LIN {X 0,Y 206.643,Z 558.739,A -85,B 0,C 180,E1 -21191.562,E2 -21191.562} C_VEL
LIN {X 0,Y 206.656,Z 558.72,A -85,B 0,C 180,E1 -21195.573,E2 -21195.573} C_VEL
LIN {X 0,Y 206.699,Z 558.712,A -85,B 0,C 180,E1 -21199.757,E2 -21199.757} C_VEL
LIN {X 0,Y 206.719,Z 558.701,A -85,B 0,C 180,E1 -21202.268,E2 -21202.268} C_VEL
LIN {X 0,Y 206.705,Z 558.728,A -85,B 0,C 180,E1 -21207.043,E2 -21207.043} C_VEL
LIN {X 0,Y 206.761,Z 558.716,A -85,B 0,C 180,E1 -21212.095,E2 -21212.095} C_VEL
LIN {X 0,Y 206.78,Z 558.717,A -85,B 0,C 180,E1 -21216.583,E2 -21216.583} C_VEL
LIN {X 0,Y 206.87,Z 558.707,A -85,B 0,C 180,E1 -21222.196,E2 -21222.196} C_VEL
LIN {X 0,Y 206.907,Z 558.71,A -85,B 0,C 180,E1 -21226.245,E2 -21226.245} C_VEL
LIN {X 0,Y 207.099,Z 558.667,A -85,B 0,C 180,E1 -21230.231,E2 -21230.231} C_VEL
LIN {X 0,Y 207.172,Z 558.672,A -85,B 0,C 180,E1 -21232.201,E2 -21232.201} C_VEL
LIN {X 0,Y 207.376,Z 558.637,A -85,B 0,C 180,E1 -21238.058,E2 -21238.058} C_VEL
LIN {X 0,Y 207.513,Z 558.637,A -85,B 0,C 180,E1 -21240,E2 -21240} C_VEL
LIN {X 0,Y 207.08,Z 558.67,A -85,B 0,C 180,E1 -21243.892,E2 -21243.892} C_VEL
LIN {X 0,Y 207.182,Z 558.674,A -85,B 0,C 180,E1 -21247.798,E2 -21247.798} C_VEL
LIN {X 0,Y 206.977,Z 558.693,A -85,B 0,C 180,E1 -21251.755,E2 -21251.755} C_VEL
LIN {X 0,Y 206.86,Z 558.701,A -85,B 0,C 180,E1 -21255.771,E2 -21255.771} C_VEL
LIN {X 0,Y 206.793,Z 558.723,A -85,B 0,C 180,E1 -21259.868,E2 -21259.868} C_VEL
LIN {X 0,Y 206.757,Z 558.732,A -85,B 0,C 180,E1 -21264.073,E2 -21264.073} C_VEL
LIN {X 0,Y 206.731,Z 558.734,A -85,B 0,C 180,E1 -21268.421,E2 -21268.421} C_VEL
LIN {X 0,Y 206.693,Z 558.739,A -85,B 0,C 180,E1 -21272.959,E2 -21272.959} C_VEL
LIN {X 0,Y 206.658,Z 558.711,A -85,B 0,C 180,E1 -21276.382,E2 -21276.382} C_VEL
LIN {X 0,Y 205.988,Z 558.801,A -85,B 0,C 180,E1 -21277.465,E2 -21277.465} C_VEL
LIN {X 0,Y 203.169,Z 559.171,A -85,B 0,C 180,E1 -21279.168,E2 -21279.168} C_VEL
LIN {X 0,Y 200.309,Z 559.522,A -85,B 0,C 180,E1 -21280.916,E2 -21280.916} C_VEL
LIN {X 0,Y 199.623,Z 559.597,A -85,B 0,C 180,E1 -21282.051,E2 -21282.051} C_VEL
LIN {X 0,Y 199.665,Z 559.81,A -85,B 0,C 180,E1 -21283.274,E2 -21283.274} C_VEL
LIN {X 0,Y 201.361,Z 565.662,A -85,B 0,C 180,E1 -21286.98,E2 -21286.98} C_VEL
LIN {X 0,Y 203.872,Z 570.231,A -85,B 0,C 180,E1 -21287.939,E2 -21287.939} C_VEL
LIN {X 0,Y 209.554,Z 580.486,A -85,B 0,C 180,E1 -21289.769,E2 -21289.769} C_VEL
LIN {X 0,Y 215.631,Z 592.995,A -85,B 0,C 180,E1 -21291.634,E2 -21291.634} C_VEL
LIN {X 0,Y 221.774,Z 607.312,A -85,B 0,C 180,E1 -21293.438,E2 -21293.438} C_VEL
LIN {X 0,Y 222.893,Z 610.666,A -85,B 0,C 180,E1 -21293.781,E2 -21293.781} C_VEL
LIN {X 0,Y 224.518,Z 623.901,A -85,B 0,C 180,E1 -21294.591,E2 -21294.591} C_VEL
LIN {X 0,Y 222.125,Z 674.384,A -85,B 0,C 180,E1 -21296.151,E2 -21296.151} C_VEL
LIN {X 0,Y 220.762,Z 687.705,A -85,B 0,C 180,E1 -21296.878,E2 -21296.878} C_VEL
LIN {X 0,Y 218.764,Z 699.996,A -85,B 0,C 180,E1 -21297.856,E2 -21297.856} C_VEL
LIN {X 0,Y 216.36,Z 712.201,A -85,B 0,C 180,E1 -21299.231,E2 -21299.231} C_VEL
LIN {X 0,Y 213.518,Z 723.76,A -85,B 0,C 180,E1 -21300.957,E2 -21300.957} C_VEL
LIN {X 0,Y 210.646,Z 734.172,A -85,B 0,C 180,E1 -21302.964,E2 -21302.964} C_VEL
LIN {X 0,Y 208.011,Z 742.689,A -85,B 0,C 180,E1 -21305.02,E2 -21305.02} C_VEL
LIN {X 0,Y 205.094,Z 751.926,A -85,B 0,C 180,E1 -21307.858,E2 -21307.858} C_VEL
LIN {X 0,Y 202.534,Z 759.353,A -85,B 0,C 180,E1 -21310.754,E2 -21310.754} C_VEL
LIN {X 0,Y 200.516,Z 765.318,A -85,B 0,C 180,E1 -21313.718,E2 -21313.718} C_VEL
LIN {X 0,Y 199.003,Z 770.036,A -85,B 0,C 180,E1 -21316.731,E2 -21316.731} C_VEL
LIN {X 0,Y 198.024,Z 773.649,A -85,B 0,C 180,E1 -21319.78,E2 -21319.78} C_VEL
LIN {X 0,Y 197.589,Z 775.512,A -85,B 0,C 180,E1 -21321.822,E2 -21321.822} C_VEL
LIN {X 0,Y 197.34,Z 776.909,A -85,B 0,C 180,E1 -21323.869,E2 -21323.869} C_VEL
LIN {X 0,Y 197.247,Z 778.517,A -85,B 0,C 180,E1 -21327.96,E2 -21327.96} C_VEL
LIN {X 0,Y 197.331,Z 778.731,A -85,B 0,C 180,E1 -21330.002,E2 -21330.002} C_VEL
LIN {X 0,Y 197.378,Z 778.507,A -85,B 0,C 180,E1 -21332.042,E2 -21332.042} C_VEL
LIN {X 0,Y 197.753,Z 777.534,A -85,B 0,C 180,E1 -21335.265,E2 -21335.265} C_VEL
LIN {X 0,Y 198.038,Z 780.359,A -85,B 0,C 180,E1 -21338.163,E2 -21338.163} C_VEL
LIN {X 0,Y 198.542,Z 781.793,A -85,B 0,C 180,E1 -21340.196,E2 -21340.196} C_VEL
LIN {X 0,Y 199.412,Z 782.694,A -85,B 0,C 180,E1 -21342.21,E2 -21342.21} C_VEL
LIN {X 0,Y 200.565,Z 783.037,A -85,B 0,C 180,E1 -21344.201,E2 -21344.201} C_VEL
LIN {X 0,Y 201.94,Z 782.915,A -85,B 0,C 180,E1 -21346.168,E2 -21346.168} C_VEL
LIN {X 0,Y 203.619,Z 782.336,A -85,B 0,C 180,E1 -21348.099,E2 -21348.099} C_VEL
LIN {X 0,Y 205.58,Z 781.284,A -85,B 0,C 180,E1 -21349.992,E2 -21349.992} C_VEL
LIN {X 0,Y 209.226,Z 778.633,A -85,B 0,C 180,E1 -21352.726,E2 -21352.726} C_VEL
LIN {X 0,Y 213.345,Z 774.775,A -85,B 0,C 180,E1 -21355.358,E2 -21355.358} C_VEL
LIN {X 0,Y 218.05,Z 769.669,A -85,B 0,C 180,E1 -21357.864,E2 -21357.864} C_VEL
LIN {X 0,Y 223.14,Z 762.876,A -85,B 0,C 180,E1 -21360.262,E2 -21360.262} C_VEL
LIN {X 0,Y 227.906,Z 755.838,A -85,B 0,C 180,E1 -21362.138,E2 -21362.138} C_VEL
LIN {X 0,Y 232.926,Z 747.036,A -85,B 0,C 180,E1 -21363.933,E2 -21363.933} C_VEL
LIN {X 0,Y 237.2,Z 738.413,A -85,B 0,C 180,E1 -21365.295,E2 -21365.295} C_VEL
LIN {X 0,Y 241.08,Z 729.19,A -85,B 0,C 180,E1 -21366.441,E2 -21366.441} C_VEL
LIN {X 0,Y 244.956,Z 717.42,A -85,B 0,C 180,E1 -21367.568,E2 -21367.568} C_VEL
LIN {X 0,Y 248.238,Z 704.464,A -85,B 0,C 180,E1 -21368.462,E2 -21368.462} C_VEL
LIN {X 0,Y 255.779,Z 670.421,A -85,B 0,C 180,E1 -21370.309,E2 -21370.309} C_VEL
LIN {X 0,Y 259.608,Z 653.752,A -85,B 0,C 180,E1 -21371.148,E2 -21371.148} C_VEL
LIN {X 0,Y 258.402,Z 653.739,A -85,B 0,C 180,E1 -21374.047,E2 -21374.047} C_VEL
LIN {X 0,Y 257.974,Z 655.742,A -85,B 0,C 180,E1 -21376.424,E2 -21376.424} C_VEL
LIN {X 0,Y 257.979,Z 658.123,A -85,B 0,C 180,E1 -21378.026,E2 -21378.026} C_VEL
LIN {X 0,Y 256.348,Z 670.35,A -85,B 0,C 180,E1 -21380.313,E2 -21380.313} C_VEL
LIN {X 0,Y 255.161,Z 681.627,A -85,B 0,C 180,E1 -21382.065,E2 -21382.065} C_VEL
LIN {X 0,Y 254.844,Z 684.003,A -85,B 0,C 180,E1 -21382.343,E2 -21382.343} C_VEL
LIN {X 0,Y 248.904,Z 711.445,A -85,B 0,C 180,E1 -21383.759,E2 -21383.759} C_VEL
LIN {X 0,Y 245.558,Z 722.701,A -85,B 0,C 180,E1 -21384.58,E2 -21384.58} C_VEL
LIN {X 0,Y 241.35,Z 733.582,A -85,B 0,C 180,E1 -21385.654,E2 -21385.654} C_VEL
LIN {X 0,Y 236.31,Z 744.211,A -85,B 0,C 180,E1 -21387.128,E2 -21387.128} C_VEL
LIN {X 0,Y 231.588,Z 752.59,A -85,B 0,C 180,E1 -21388.623,E2 -21388.623} C_VEL
LIN {X 0,Y 226.898,Z 759.605,A -85,B 0,C 180,E1 -21390.291,E2 -21390.291} C_VEL
LIN {X 0,Y 222.191,Z 765.752,A -85,B 0,C 180,E1 -21392.189,E2 -21392.189} C_VEL
LIN {X 0,Y 217.858,Z 770.669,A -85,B 0,C 180,E1 -21394.183,E2 -21394.183} C_VEL
LIN {X 0,Y 213.113,Z 775.192,A -85,B 0,C 180,E1 -21396.688,E2 -21396.688} C_VEL
LIN {X 0,Y 210.249,Z 777.424,A -85,B 0,C 180,E1 -21398.426,E2 -21398.426} C_VEL
LIN {X 0,Y 207.601,Z 779.05,A -85,B 0,C 180,E1 -21400.212,E2 -21400.212} C_VEL
LIN {X 0,Y 205.294,Z 780.132,A -85,B 0,C 180,E1 -21402.055,E2 -21402.055} C_VEL
LIN {X 0,Y 203.381,Z 780.726,A -85,B 0,C 180,E1 -21403.952,E2 -21403.952} C_VEL
LIN {X 0,Y 201.76,Z 780.834,A -85,B 0,C 180,E1 -21405.887,E2 -21405.887} C_VEL
LIN {X 0,Y 200.399,Z 780.44,A -85,B 0,C 180,E1 -21407.853,E2 -21407.853} C_VEL
LIN {X 0,Y 199.338,Z 779.484,A -85,B 0,C 180,E1 -21409.847,E2 -21409.847} C_VEL
LIN {X 0,Y 198.172,Z 776.715,A -85,B 0,C 180,E1 -21413.225,E2 -21413.225} C_VEL
LIN {X 0,Y 197.867,Z 773.43,A -85,B 0,C 180,E1 -21415.926,E2 -21415.926} C_VEL
LIN {X 0,Y 197.89,Z 768.393,A -85,B 0,C 180,E1 -21418.983,E2 -21418.983} C_VEL
LIN {X 0,Y 198.227,Z 761.55,A -85,B 0,C 180,E1 -21422.032,E2 -21422.032} C_VEL
LIN {X 0,Y 198.413,Z 755.716,A -85,B 0,C 180,E1 -21424.062,E2 -21424.062} C_VEL
LIN {X 0,Y 198.864,Z 747.227,A -85,B 0,C 180,E1 -21426.477,E2 -21426.477} C_VEL
LIN {X 0,Y 199.278,Z 738.663,A -85,B 0,C 180,E1 -21428.38,E2 -21428.38} C_VEL
LIN {X 0,Y 199.692,Z 728.558,A -85,B 0,C 180,E1 -21430.135,E2 -21430.135} C_VEL
LIN {X 0,Y 200.238,Z 717.043,A -85,B 0,C 180,E1 -21431.643,E2 -21431.643} C_VEL
LIN {X 0,Y 200.585,Z 705.7,A -85,B 0,C 180,E1 -21432.714,E2 -21432.714} C_VEL
LIN {X 0,Y 201.604,Z 660.067,A -85,B 0,C 180,E1 -21435.674,E2 -21435.674} C_VEL
LIN {X 0,Y 200.19,Z 633.11,A -85,B 0,C 180,E1 -21437.362,E2 -21437.362} C_VEL
LIN {X 0,Y 200.23,Z 631.57,A -85,B 0,C 180,E1 -21437.622,E2 -21437.622} C_VEL
LIN {X 0,Y 202.024,Z 611.253,A -85,B 0,C 180,E1 -21443.04,E2 -21443.04} C_VEL
LIN {X 0,Y 204.085,Z 591.489,A -85,B 0,C 180,E1 -21448.262,E2 -21448.262} C_VEL
LIN {X 0,Y 204.812,Z 584.337,A -85,B 0,C 180,E1 -21450.145,E2 -21450.145} C_VEL
LIN {X 0,Y 201.716,Z 569.092,A -85,B 0,C 180,E1 -21454.413,E2 -21454.413} C_VEL
LIN {X 0,Y 199.808,Z 559.78,A -85,B 0,C 180,E1 -21457.157,E2 -21457.157} C_VEL
LIN {X 0,Y 199.581,Z 559.561,A -85,B 0,C 180,E1 -21462.31,E2 -21462.31} C_VEL
LIN {X 0,Y 199.677,Z 559.818,A -85,B 0,C 180,E1 -21466.585,E2 -21466.585} C_VEL
LIN {X 0,Y 199.952,Z 560.952,A -85,B 0,C 180,E1 -21466.993,E2 -21466.993} C_VEL
LIN {X 0,Y 201.638,Z 563.728,A -85,B 0,C 180,E1 -21467.594,E2 -21467.594} C_VEL
LIN {X 0,Y 202.715,Z 565.008,A -85,B 0,C 180,E1 -21467.934,E2 -21467.934} C_VEL
LIN {X 0,Y 205.044,Z 568.455,A -85,B 0,C 180,E1 -21468.681,E2 -21468.681} C_VEL
LIN {X 0,Y 213.235,Z 581.719,A -85,B 0,C 180,E1 -21471.169,E2 -21471.169} C_VEL
LIN {X 0,Y 220.429,Z 596.663,A -85,B 0,C 180,E1 -21473.27,E2 -21473.27} C_VEL
LIN {X 0,Y 225.025,Z 607.882,A -85,B 0,C 180,E1 -21474.578,E2 -21474.578} C_VEL
LIN {X 0,Y 222.424,Z 664.276,A -85,B 0,C 180,E1 -21476.339,E2 -21476.339} C_VEL
LIN {X 0,Y 221.083,Z 677.457,A -85,B 0,C 180,E1 -21477.073,E2 -21477.073} C_VEL
LIN {X 0,Y 219.394,Z 689.53,A -85,B 0,C 180,E1 -21478.09,E2 -21478.09} C_VEL
LIN {X 0,Y 217.347,Z 700.817,A -85,B 0,C 180,E1 -21479.382,E2 -21479.382} C_VEL
LIN {X 0,Y 214.559,Z 712.45,A -85,B 0,C 180,E1 -21481.107,E2 -21481.107} C_VEL
LIN {X 0,Y 211.759,Z 722.896,A -85,B 0,C 180,E1 -21483.114,E2 -21483.114} C_VEL
LIN {X 0,Y 209.106,Z 732.051,A -85,B 0,C 180,E1 -21485.345,E2 -21485.345} C_VEL
LIN {X 0,Y 206.368,Z 740.665,A -85,B 0,C 180,E1 -21487.998,E2 -21487.998} C_VEL
LIN {X 0,Y 203.743,Z 748.068,A -85,B 0,C 180,E1 -21490.869,E2 -21490.869} C_VEL
LIN {X 0,Y 201.639,Z 754.008,A -85,B 0,C 180,E1 -21493.808,E2 -21493.808} C_VEL
LIN {X 0,Y 199.942,Z 758.7,A -85,B 0,C 180,E1 -21496.791,E2 -21496.791} C_VEL
LIN {X 0,Y 198.741,Z 762.283,A -85,B 0,C 180,E1 -21499.814,E2 -21499.814} C_VEL
LIN {X 0,Y 198.164,Z 764.133,A -85,B 0,C 180,E1 -21501.843,E2 -21501.843} C_VEL
LIN {X 0,Y 197.671,Z 765.903,A -85,B 0,C 180,E1 -21504.575,E2 -21504.575} C_VEL
LIN {X 0,Y 197.407,Z 767.121,A -85,B 0,C 180,E1 -21507.958,E2 -21507.958} C_VEL
LIN {X 0,Y 197.401,Z 767.348,A -85,B 0,C 180,E1 -21509.998,E2 -21509.998} C_VEL
LIN {X 0,Y 197.406,Z 767.155,A -85,B 0,C 180,E1 -21512.038,E2 -21512.038} C_VEL
LIN {X 0,Y 197.669,Z 765.987,A -85,B 0,C 180,E1 -21515.419,E2 -21515.419} C_VEL
LIN {X 0,Y 198.162,Z 764.251,A -85,B 0,C 180,E1 -21518.154,E2 -21518.154} C_VEL
LIN {X 0,Y 199.056,Z 761.381,A -85,B 0,C 180,E1 -21521.195,E2 -21521.195} C_VEL
LIN {X 0,Y 200.419,Z 757.487,A -85,B 0,C 180,E1 -21524.207,E2 -21524.207} C_VEL
LIN {X 0,Y 202.212,Z 752.468,A -85,B 0,C 180,E1 -21527.181,E2 -21527.181} C_VEL
LIN {X 0,Y 204.465,Z 746.143,A -85,B 0,C 180,E1 -21530.102,E2 -21530.102} C_VEL
LIN {X 0,Y 207.302,Z 738.221,A -85,B 0,C 180,E1 -21532.945,E2 -21532.945} C_VEL
LIN {X 0,Y 209.92,Z 729.627,A -85,B 0,C 180,E1 -21535.424,E2 -21535.424} C_VEL
LIN {X 0,Y 212.584,Z 720.302,A -85,B 0,C 180,E1 -21537.568,E2 -21537.568} C_VEL
LIN {X 0,Y 215.469,Z 709.206,A -85,B 0,C 180,E1 -21539.558,E2 -21539.558} C_VEL
LIN {X 0,Y 217.881,Z 698.322,A -85,B 0,C 180,E1 -21541.069,E2 -21541.069} C_VEL
LIN {X 0,Y 220.02,Z 686.282,A -85,B 0,C 180,E1 -21542.344,E2 -21542.344} C_VEL
LIN {X 0,Y 221.684,Z 673.728,A -85,B 0,C 180,E1 -21543.299,E2 -21543.299} C_VEL
LIN {X 0,Y 222.779,Z 660.908,A -85,B 0,C 180,E1 -21543.918,E2 -21543.918} C_VEL
LIN {X 0,Y 225.154,Z 608.113,A -85,B 0,C 180,E1 -21545.54,E2 -21545.54} C_VEL
LIN {X 0,Y 219.131,Z 593.766,A -85,B 0,C 180,E1 -21547.258,E2 -21547.258} C_VEL
LIN {X 0,Y 212.658,Z 580.606,A -85,B 0,C 180,E1 -21549.166,E2 -21549.166} C_VEL
LIN {X 0,Y 205.028,Z 568.468,A -85,B 0,C 180,E1 -21551.492,E2 -21551.492} C_VEL
LIN {X 0,Y 202.812,Z 565.309,A -85,B 0,C 180,E1 -21552.2,E2 -21552.2} C_VEL
LIN {X 0,Y 202.07,Z 564.19,A -85,B 0,C 180,E1 -21552.445,E2 -21552.445} C_VEL
LIN {X 0,Y 200.158,Z 561.683,A -85,B 0,C 180,E1 -21553.072,E2 -21553.072} C_VEL
LIN {X 0,Y 199.577,Z 559.608,A -85,B 0,C 180,E1 -21553.387,E2 -21553.387} C_VEL
LIN {X 0,Y 199.615,Z 559.621,A -85,B 0,C 180,E1 -21558.014,E2 -21558.014} C_VEL
LIN {X 0,Y 199.673,Z 559.577,A -85,B 0,C 180,E1 -21560.742,E2 -21560.742} C_VEL
LIN {X 0,Y 199.631,Z 559.619,A -85,B 0,C 180,E1 -21565.717,E2 -21565.717} C_VEL
LIN {X 0,Y 199.699,Z 559.6,A -85,B 0,C 180,E1 -21568.136,E2 -21568.136} C_VEL
LIN {X 0,Y 199.681,Z 559.598,A -85,B 0,C 180,E1 -21572.771,E2 -21572.771} C_VEL
LIN {X 0,Y 199.732,Z 559.59,A -85,B 0,C 180,E1 -21577.228,E2 -21577.228} C_VEL
LIN {X 0,Y 199.832,Z 559.587,A -85,B 0,C 180,E1 -21581.721,E2 -21581.721} C_VEL
LIN {X 0,Y 199.841,Z 559.584,A -85,B 0,C 180,E1 -21585.749,E2 -21585.749} C_VEL
LIN {X 0,Y 200.064,Z 559.543,A -85,B 0,C 180,E1 -21589.884,E2 -21589.884} C_VEL
LIN {X 0,Y 200.033,Z 559.567,A -85,B 0,C 180,E1 -21593.95,E2 -21593.95} C_VEL
LIN {X 0,Y 200.316,Z 559.516,A -85,B 0,C 180,E1 -21597.989,E2 -21597.989} C_VEL
LIN {X 0,Y 200.477,Z 559.514,A -85,B 0,C 180,E1 -21600,E2 -21600} C_VEL
LIN {X 0,Y 200.026,Z 559.549,A -85,B 0,C 180,E1 -21604.029,E2 -21604.029} C_VEL
LIN {X 0,Y 200.126,Z 559.552,A -85,B 0,C 180,E1 -21608.075,E2 -21608.075} C_VEL
LIN {X 0,Y 199.908,Z 559.577,A -85,B 0,C 180,E1 -21612.177,E2 -21612.177} C_VEL
LIN {X 0,Y 199.799,Z 559.58,A -85,B 0,C 180,E1 -21616.344,E2 -21616.344} C_VEL
LIN {X 0,Y 199.818,Z 559.594,A -85,B 0,C 180,E1 -21618.454,E2 -21618.454} C_VEL
LIN {X 0,Y 199.731,Z 559.605,A -85,B 0,C 180,E1 -21623.818,E2 -21623.818} C_VEL
LIN {X 0,Y 199.702,Z 559.608,A -85,B 0,C 180,E1 -21628.385,E2 -21628.385} C_VEL
LIN {X 0,Y 199.666,Z 559.611,A -85,B 0,C 180,E1 -21632.356,E2 -21632.356} C_VEL
LIN {X 0,Y 199.638,Z 559.584,A -85,B 0,C 180,E1 -21636.76,E2 -21636.76} C_VEL
LIN {X 0,Y 199.669,Z 559.61,A -85,B 0,C 180,E1 -21639.314,E2 -21639.314} C_VEL
LIN {X 0,Y 199.623,Z 559.597,A -85,B 0,C 180,E1 -21642.051,E2 -21642.051} C_VEL
LIN {X 0,Y 199.313,Z 560.282,A -85,B 0,C 180,E1 -21642.984,E2 -21642.984} C_VEL
LIN {X 0,Y 198.369,Z 562.793,A -85,B 0,C 180,E1 -21644.129,E2 -21644.129} C_VEL
LIN {X 0,Y 197.419,Z 566.85,A -85,B 0,C 180,E1 -21645.236,E2 -21645.236} C_VEL
LIN {X 0,Y 197.48,Z 570.795,A -85,B 0,C 180,E1 -21646.115,E2 -21646.115} C_VEL
LIN {X 0,Y 198.563,Z 573.421,A -85,B 0,C 180,E1 -21646.705,E2 -21646.705} C_VEL
LIN {X 0,Y 203.685,Z 582.425,A -85,B 0,C 180,E1 -21648.456,E2 -21648.456} C_VEL
LIN {X 0,Y 210.102,Z 595.374,A -85,B 0,C 180,E1 -21650.541,E2 -21650.541} C_VEL
LIN {X 0,Y 216.727,Z 611.183,A -85,B 0,C 180,E1 -21652.607,E2 -21652.607} C_VEL
LIN {X 0,Y 217.406,Z 613.834,A -85,B 0,C 180,E1 -21652.85,E2 -21652.85} C_VEL
LIN {X 0,Y 218.724,Z 624.414,A -85,B 0,C 180,E1 -21653.533,E2 -21653.533} C_VEL
LIN {X 0,Y 216.213,Z 675.123,A -85,B 0,C 180,E1 -21655.151,E2 -21655.151} C_VEL
LIN {X 0,Y 214.664,Z 688.967,A -85,B 0,C 180,E1 -21655.945,E2 -21655.945} C_VEL
LIN {X 0,Y 212.576,Z 700.905,A -85,B 0,C 180,E1 -21656.943,E2 -21656.943} C_VEL
LIN {X 0,Y 209.92,Z 713.586,A -85,B 0,C 180,E1 -21658.461,E2 -21658.461} C_VEL
LIN {X 0,Y 206.973,Z 724.852,A -85,B 0,C 180,E1 -21660.226,E2 -21660.226} C_VEL
LIN {X 0,Y 203.997,Z 735.005,A -85,B 0,C 180,E1 -21662.286,E2 -21662.286} C_VEL
LIN {X 0,Y 201.01,Z 744.156,A -85,B 0,C 180,E1 -21664.642,E2 -21664.642} C_VEL
LIN {X 0,Y 198.218,Z 752.585,A -85,B 0,C 180,E1 -21667.396,E2 -21667.396} C_VEL
LIN {X 0,Y 195.461,Z 760.265,A -85,B 0,C 180,E1 -21670.576,E2 -21670.576} C_VEL
LIN {X 0,Y 193.045,Z 766.806,A -85,B 0,C 180,E1 -21674.157,E2 -21674.157} C_VEL
LIN {X 0,Y 191.66,Z 771.143,A -85,B 0,C 180,E1 -21677.292,E2 -21677.292} C_VEL
LIN {X 0,Y 191.013,Z 773.445,A -85,B 0,C 180,E1 -21679.401,E2 -21679.401} C_VEL
LIN {X 0,Y 190.538,Z 775.307,A -85,B 0,C 180,E1 -21681.518,E2 -21681.518} C_VEL
LIN {X 0,Y 190.278,Z 776.705,A -85,B 0,C 180,E1 -21683.64,E2 -21683.64} C_VEL
LIN {X 0,Y 190.155,Z 778.312,A -85,B 0,C 180,E1 -21687.884,E2 -21687.884} C_VEL
LIN {X 0,Y 190.236,Z 778.526,A -85,B 0,C 180,E1 -21690.002,E2 -21690.002} C_VEL
LIN {X 0,Y 190.291,Z 778.302,A -85,B 0,C 180,E1 -21692.118,E2 -21692.118} C_VEL
LIN {X 0,Y 190.844,Z 777.039,A -85,B 0,C 180,E1 -21696.12,E2 -21696.12} C_VEL
LIN {X 0,Y 191.058,Z 779.447,A -85,B 0,C 180,E1 -21698.463,E2 -21698.463} C_VEL
LIN {X 0,Y 191.594,Z 781.043,A -85,B 0,C 180,E1 -21700.57,E2 -21700.57} C_VEL
LIN {X 0,Y 192.511,Z 782.153,A -85,B 0,C 180,E1 -21702.655,E2 -21702.655} C_VEL
LIN {X 0,Y 193.704,Z 782.81,A -85,B 0,C 180,E1 -21704.715,E2 -21704.715} C_VEL
LIN {X 0,Y 195.147,Z 783.008,A -85,B 0,C 180,E1 -21706.747,E2 -21706.747} C_VEL
LIN {X 0,Y 196.885,Z 782.666,A -85,B 0,C 180,E1 -21708.741,E2 -21708.741} C_VEL
LIN {X 0,Y 198.942,Z 781.819,A -85,B 0,C 180,E1 -21710.689,E2 -21710.689} C_VEL
LIN {X 0,Y 201.489,Z 780.484,A -85,B 0,C 180,E1 -21712.564,E2 -21712.564} C_VEL
LIN {X 0,Y 205.568,Z 777.591,A -85,B 0,C 180,E1 -21715.301,E2 -21715.301} C_VEL
LIN {X 0,Y 210.343,Z 773.457,A -85,B 0,C 180,E1 -21717.891,E2 -21717.891} C_VEL
LIN {X 0,Y 215.547,Z 767.896,A -85,B 0,C 180,E1 -21720.359,E2 -21720.359} C_VEL
LIN {X 0,Y 220.307,Z 762.035,A -85,B 0,C 180,E1 -21722.301,E2 -21722.301} C_VEL
LIN {X 0,Y 226.49,Z 753.294,A -85,B 0,C 180,E1 -21724.494,E2 -21724.494} C_VEL
LIN {X 0,Y 231.437,Z 744.927,A -85,B 0,C 180,E1 -21726.042,E2 -21726.042} C_VEL
LIN {X 0,Y 236.629,Z 734.698,A -85,B 0,C 180,E1 -21727.509,E2 -21727.509} C_VEL
LIN {X 0,Y 240.761,Z 724.592,A -85,B 0,C 180,E1 -21728.607,E2 -21728.607} C_VEL
LIN {X 0,Y 244.395,Z 713.469,A -85,B 0,C 180,E1 -21729.514,E2 -21729.514} C_VEL
LIN {X 0,Y 248.288,Z 697.651,A -85,B 0,C 180,E1 -21730.488,E2 -21730.488} C_VEL
LIN {X 0,Y 254.976,Z 669.376,A -85,B 0,C 180,E1 -21731.936,E2 -21731.936} C_VEL
LIN {X 0,Y 257.137,Z 660.432,A -85,B 0,C 180,E1 -21732.442,E2 -21732.442} C_VEL
LIN {X 0,Y 256.503,Z 660.855,A -85,B 0,C 180,E1 -21734.367,E2 -21734.367} C_VEL
LIN {X 0,Y 256.112,Z 663.035,A -85,B 0,C 180,E1 -21736.573,E2 -21736.573} C_VEL
LIN {X 0,Y 256.07,Z 663.953,A -85,B 0,C 180,E1 -21737.123,E2 -21737.123} C_VEL
LIN {X 0,Y 254.151,Z 675.571,A -85,B 0,C 180,E1 -21739.301,E2 -21739.301} C_VEL
LIN {X 0,Y 252.699,Z 685.678,A -85,B 0,C 180,E1 -21740.859,E2 -21740.859} C_VEL
LIN {X 0,Y 246.939,Z 711.044,A -85,B 0,C 180,E1 -21742.144,E2 -21742.144} C_VEL
LIN {X 0,Y 243.455,Z 722.275,A -85,B 0,C 180,E1 -21742.943,E2 -21742.943} C_VEL
LIN {X 0,Y 239.627,Z 731.754,A -85,B 0,C 180,E1 -21743.826,E2 -21743.826} C_VEL
LIN {X 0,Y 234.811,Z 741.897,A -85,B 0,C 180,E1 -21745.081,E2 -21745.081} C_VEL
LIN {X 0,Y 229.638,Z 750.729,A -85,B 0,C 180,E1 -21746.572,E2 -21746.572} C_VEL
LIN {X 0,Y 224.314,Z 758.556,A -85,B 0,C 180,E1 -21748.279,E2 -21748.279} C_VEL
LIN {X 0,Y 219.033,Z 765.044,A -85,B 0,C 180,E1 -21750.176,E2 -21750.176} C_VEL
LIN {X 0,Y 215.229,Z 769.152,A -85,B 0,C 180,E1 -21751.739,E2 -21751.739} C_VEL
LIN {X 0,Y 209.958,Z 774.044,A -85,B 0,C 180,E1 -21754.205,E2 -21754.205} C_VEL
LIN {X 0,Y 206.715,Z 776.508,A -85,B 0,C 180,E1 -21755.922,E2 -21755.922} C_VEL
LIN {X 0,Y 203.717,Z 778.405,A -85,B 0,C 180,E1 -21757.698,E2 -21757.698} C_VEL
LIN {X 0,Y 200.973,Z 779.797,A -85,B 0,C 180,E1 -21759.531,E2 -21759.531} C_VEL
LIN {X 0,Y 198.596,Z 780.66,A -85,B 0,C 180,E1 -21761.428,E2 -21761.428} C_VEL
LIN {X 0,Y 196.589,Z 780.953,A -85,B 0,C 180,E1 -21763.382,E2 -21763.382} C_VEL
LIN {X 0,Y 194.888,Z 780.736,A -85,B 0,C 180,E1 -21765.379,E2 -21765.379} C_VEL
LIN {X 0,Y 193.494,Z 780.049,A -85,B 0,C 180,E1 -21767.413,E2 -21767.413} C_VEL
LIN {X 0,Y 192.389,Z 778.886,A -85,B 0,C 180,E1 -21769.476,E2 -21769.476} C_VEL
LIN {X 0,Y 191.6,Z 777.235,A -85,B 0,C 180,E1 -21771.563,E2 -21771.563} C_VEL
LIN {X 0,Y 190.968,Z 773.747,A -85,B 0,C 180,E1 -21774.607,E2 -21774.607} C_VEL
LIN {X 0,Y 190.904,Z 768.638,A -85,B 0,C 180,E1 -21777.89,E2 -21777.89} C_VEL
LIN {X 0,Y 191.188,Z 762.049,A -85,B 0,C 180,E1 -21781.053,E2 -21781.053} C_VEL
LIN {X 0,Y 191.466,Z 756.372,A -85,B 0,C 180,E1 -21783.156,E2 -21783.156} C_VEL
LIN {X 0,Y 191.885,Z 747.559,A -85,B 0,C 180,E1 -21785.781,E2 -21785.781} C_VEL
LIN {X 0,Y 192.283,Z 738.777,A -85,B 0,C 180,E1 -21787.82,E2 -21787.82} C_VEL
LIN {X 0,Y 192.664,Z 729.114,A -85,B 0,C 180,E1 -21789.595,E2 -21789.595} C_VEL
LIN {X 0,Y 193.165,Z 718.19,A -85,B 0,C 180,E1 -21791.144,E2 -21791.144} C_VEL
LIN {X 0,Y 193.579,Z 706.742,A -85,B 0,C 180,E1 -21792.315,E2 -21792.315} C_VEL
LIN {X 0,Y 194.525,Z 659.858,A -85,B 0,C 180,E1 -21795.52,E2 -21795.52} C_VEL
LIN {X 0,Y 193.109,Z 633.055,A -85,B 0,C 180,E1 -21797.268,E2 -21797.268} C_VEL
LIN {X 0,Y 193.106,Z 631.825,A -85,B 0,C 180,E1 -21797.473,E2 -21797.473} C_VEL
LIN {X 0,Y 195.009,Z 610.41,A -85,B 0,C 180,E1 -21803.356,E2 -21803.356} C_VEL
LIN {X 0,Y 197.294,Z 589.517,A -85,B 0,C 180,E1 -21809.036,E2 -21809.036} C_VEL
LIN {X 0,Y 197.717,Z 584.862,A -85,B 0,C 180,E1 -21810.297,E2 -21810.297} C_VEL
LIN {X 0,Y 194.737,Z 570.374,A -85,B 0,C 180,E1 -21814.456,E2 -21814.456} C_VEL
LIN {X 0,Y 192.739,Z 560.681,A -85,B 0,C 180,E1 -21817.382,E2 -21817.382} C_VEL
LIN {X 0,Y 192.522,Z 560.439,A -85,B 0,C 180,E1 -21823.103,E2 -21823.103} C_VEL
LIN {X 0,Y 192.607,Z 560.793,A -85,B 0,C 180,E1 -21824.646,E2 -21824.646} C_VEL
LIN {X 0,Y 192.938,Z 561.931,A -85,B 0,C 180,E1 -21825.055,E2 -21825.055} C_VEL
LIN {X 0,Y 194.545,Z 564.576,A -85,B 0,C 180,E1 -21825.683,E2 -21825.683} C_VEL
LIN {X 0,Y 195.73,Z 565.827,A -85,B 0,C 180,E1 -21826.086,E2 -21826.086} C_VEL
LIN {X 0,Y 198.122,Z 569.451,A -85,B 0,C 180,E1 -21826.931,E2 -21826.931} C_VEL
LIN {X 0,Y 204.033,Z 578.563,A -85,B 0,C 180,E1 -21828.895,E2 -21828.895} C_VEL
LIN {X 0,Y 208.753,Z 586.374,A -85,B 0,C 180,E1 -21830.369,E2 -21830.369} C_VEL
LIN {X 0,Y 215.819,Z 601.464,A -85,B 0,C 180,E1 -21832.542,E2 -21832.542} C_VEL
LIN {X 0,Y 219.224,Z 609.857,A -85,B 0,C 180,E1 -21833.562,E2 -21833.562} C_VEL
LIN {X 0,Y 216.633,Z 663.621,A -85,B 0,C 180,E1 -21835.259,E2 -21835.259} C_VEL
LIN {X 0,Y 215.217,Z 677.201,A -85,B 0,C 180,E1 -21836.013,E2 -21836.013} C_VEL
LIN {X 0,Y 213.422,Z 689.741,A -85,B 0,C 180,E1 -21837.087,E2 -21837.087} C_VEL
LIN {X 0,Y 211.287,Z 701.026,A -85,B 0,C 180,E1 -21838.405,E2 -21838.405} C_VEL
LIN {X 0,Y 208.37,Z 712.659,A -85,B 0,C 180,E1 -21840.164,E2 -21840.164} C_VEL
LIN {X 0,Y 205.461,Z 723.104,A -85,B 0,C 180,E1 -21842.22,E2 -21842.22} C_VEL
LIN {X 0,Y 202.491,Z 732.809,A -85,B 0,C 180,E1 -21844.664,E2 -21844.664} C_VEL
LIN {X 0,Y 199.794,Z 740.872,A -85,B 0,C 180,E1 -21847.234,E2 -21847.234} C_VEL
LIN {X 0,Y 197.025,Z 748.276,A -85,B 0,C 180,E1 -21850.19,E2 -21850.19} C_VEL
LIN {X 0,Y 194.823,Z 754.215,A -85,B 0,C 180,E1 -21853.225,E2 -21853.225} C_VEL
LIN {X 0,Y 193.033,Z 758.906,A -85,B 0,C 180,E1 -21856.309,E2 -21856.309} C_VEL
LIN {X 0,Y 191.748,Z 762.489,A -85,B 0,C 180,E1 -21859.438,E2 -21859.438} C_VEL
LIN {X 0,Y 191.127,Z 764.339,A -85,B 0,C 180,E1 -21861.54,E2 -21861.54} C_VEL
LIN {X 0,Y 190.569,Z 766.285,A -85,B 0,C 180,E1 -21864.709,E2 -21864.709} C_VEL
LIN {X 0,Y 190.317,Z 767.325,A -85,B 0,C 180,E1 -21867.882,E2 -21867.882} C_VEL
LIN {X 0,Y 190.306,Z 767.553,A -85,B 0,C 180,E1 -21869.998,E2 -21869.998} C_VEL
LIN {X 0,Y 190.316,Z 767.36,A -85,B 0,C 180,E1 -21872.114,E2 -21872.114} C_VEL
LIN {X 0,Y 190.721,Z 765.81,A -85,B 0,C 180,E1 -21876.345,E2 -21876.345} C_VEL
LIN {X 0,Y 191.125,Z 764.455,A -85,B 0,C 180,E1 -21878.456,E2 -21878.456} C_VEL
LIN {X 0,Y 192.098,Z 761.585,A -85,B 0,C 180,E1 -21881.606,E2 -21881.606} C_VEL
LIN {X 0,Y 193.538,Z 757.691,A -85,B 0,C 180,E1 -21884.724,E2 -21884.724} C_VEL
LIN {X 0,Y 195.431,Z 752.671,A -85,B 0,C 180,E1 -21887.797,E2 -21887.797} C_VEL
LIN {X 0,Y 197.816,Z 746.346,A -85,B 0,C 180,E1 -21890.808,E2 -21890.808} C_VEL
LIN {X 0,Y 200.779,Z 738.424,A -85,B 0,C 180,E1 -21893.735,E2 -21893.735} C_VEL
LIN {X 0,Y 203.426,Z 730.126,A -85,B 0,C 180,E1 -21896.204,E2 -21896.204} C_VEL
LIN {X 0,Y 206.328,Z 720.502,A -85,B 0,C 180,E1 -21898.479,E2 -21898.479} C_VEL
LIN {X 0,Y 209.343,Z 709.406,A -85,B 0,C 180,E1 -21900.513,E2 -21900.513} C_VEL
LIN {X 0,Y 211.831,Z 698.521,A -85,B 0,C 180,E1 -21902.06,E2 -21902.06} C_VEL
LIN {X 0,Y 214.048,Z 686.479,A -85,B 0,C 180,E1 -21903.362,E2 -21903.362} C_VEL
LIN {X 0,Y 215.832,Z 673.549,A -85,B 0,C 180,E1 -21904.354,E2 -21904.354} C_VEL
LIN {X 0,Y 216.992,Z 659.971,A -85,B 0,C 180,E1 -21905.005,E2 -21905.005} C_VEL
LIN {X 0,Y 219.364,Z 610.045,A -85,B 0,C 180,E1 -21906.557,E2 -21906.557} C_VEL
LIN {X 0,Y 212.653,Z 594.364,A -85,B 0,C 180,E1 -21908.581,E2 -21908.581} C_VEL
LIN {X 0,Y 207.408,Z 583.914,A -85,B 0,C 180,E1 -21910.218,E2 -21910.218} C_VEL
LIN {X 0,Y 200.592,Z 573.182,A -85,B 0,C 180,E1 -21912.405,E2 -21912.405} C_VEL
LIN {X 0,Y 197.382,Z 568.633,A -85,B 0,C 180,E1 -21913.491,E2 -21913.491} C_VEL
LIN {X 0,Y 195.174,Z 565.175,A -85,B 0,C 180,E1 -21914.288,E2 -21914.288} C_VEL
LIN {X 0,Y 193.221,Z 562.728,A -85,B 0,C 180,E1 -21914.985,E2 -21914.985} C_VEL
LIN {X 0,Y 192.56,Z 560.474,A -85,B 0,C 180,E1 -21915.352,E2 -21915.352} C_VEL
LIN {X 0,Y 192.571,Z 560.467,A -85,B 0,C 180,E1 -21920.029,E2 -21920.029} C_VEL
LIN {X 0,Y 192.597,Z 560.486,A -85,B 0,C 180,E1 -21924.278,E2 -21924.278} C_VEL
LIN {X 0,Y 192.603,Z 560.492,A -85,B 0,C 180,E1 -21929.279,E2 -21929.279} C_VEL
LIN {X 0,Y 192.659,Z 560.474,A -85,B 0,C 180,E1 -21931.691,E2 -21931.691} C_VEL
LIN {X 0,Y 192.7,Z 560.472,A -85,B 0,C 180,E1 -21936.348,E2 -21936.348} C_VEL
LIN {X 0,Y 192.775,Z 560.468,A -85,B 0,C 180,E1 -21941.413,E2 -21941.413} C_VEL
LIN {X 0,Y 192.846,Z 560.462,A -85,B 0,C 180,E1 -21947.369,E2 -21947.369} C_VEL
LIN {X 0,Y 193.062,Z 560.422,A -85,B 0,C 180,E1 -21951.627,E2 -21951.627} C_VEL
LIN {X 0,Y 193.258,Z 560.394,A -85,B 0,C 180,E1 -21957.916,E2 -21957.916} C_VEL
LIN {X 0,Y 193.44,Z 560.39,A -85,B 0,C 180,E1 -21960,E2 -21960} C_VEL
LIN {X 0,Y 192.973,Z 560.427,A -85,B 0,C 180,E1 -21964.177,E2 -21964.177} C_VEL
LIN {X 0,Y 193.073,Z 560.426,A -85,B 0,C 180,E1 -21968.372,E2 -21968.372} C_VEL
LIN {X 0,Y 192.847,Z 560.462,A -85,B 0,C 180,E1 -21972.63,E2 -21972.63} C_VEL
LIN {X 0,Y 192.775,Z 560.472,A -85,B 0,C 180,E1 -21978.587,E2 -21978.587} C_VEL
LIN {X 0,Y 192.658,Z 560.488,A -85,B 0,C 180,E1 -21984.225,E2 -21984.225} C_VEL
LIN {X 0,Y 192.638,Z 560.491,A -85,B 0,C 180,E1 -21988.89,E2 -21988.89} C_VEL
LIN {X 0,Y 192.591,Z 560.497,A -85,B 0,C 180,E1 -21993.187,E2 -21993.187} C_VEL
LIN {X 0,Y 192.59,Z 560.474,A -85,B 0,C 180,E1 -21998.343,E2 -21998.343} C_VEL
LIN {X 0,Y 192.601,Z 560.624,A -85,B 0,C 180,E1 -22001.661,E2 -22001.661} C_VEL
LIN {X 0,Y 193.957,Z 565.253,A -85,B 0,C 180,E1 -22004.866,E2 -22004.866} C_VEL
LIN {X 0,Y 196.049,Z 569.224,A -85,B 0,C 180,E1 -22005.805,E2 -22005.805} C_VEL
LIN {X 0,Y 198.139,Z 572.599,A -85,B 0,C 180,E1 -22006.55,E2 -22006.55} C_VEL
LIN {X 0,Y 198.563,Z 573.421,A -85,B 0,C 180,E1 -22006.705,E2 -22006.705} C_VEL
LIN {X 0,Y 200.178,Z 576.38,A -85,B 0,C 180,E1 -22007.278,E2 -22007.278} C_VEL
LIN {X 0,Y 201.368,Z 579.745,A -85,B 0,C 180,E1 -22007.747,E2 -22007.747} C_VEL
LIN {X 0,Y 202.922,Z 587.097,A -85,B 0,C 180,E1 -22008.482,E2 -22008.482} C_VEL
LIN {X 0,Y 204.221,Z 594.738,A -85,B 0,C 180,E1 -22009.15,E2 -22009.15} C_VEL
LIN {X 0,Y 205.688,Z 600.191,A -85,B 0,C 180,E1 -22009.744,E2 -22009.744} C_VEL
LIN {X 0,Y 206.365,Z 601.888,A -85,B 0,C 180,E1 -22009.977,E2 -22009.977} C_VEL
LIN {X 0,Y 211.681,Z 614.929,A -85,B 0,C 180,E1 -22011.721,E2 -22011.721} C_VEL
LIN {X 0,Y 212.97,Z 626.151,A -85,B 0,C 180,E1 -22012.46,E2 -22012.46} C_VEL
LIN {X 0,Y 210.473,Z 674.062,A -85,B 0,C 180,E1 -22013.999,E2 -22013.999} C_VEL
LIN {X 0,Y 209.064,Z 687.047,A -85,B 0,C 180,E1 -22014.734,E2 -22014.734} C_VEL
LIN {X 0,Y 206.907,Z 699.602,A -85,B 0,C 180,E1 -22015.768,E2 -22015.768} C_VEL
LIN {X 0,Y 204.262,Z 711.801,A -85,B 0,C 180,E1 -22017.189,E2 -22017.189} C_VEL
LIN {X 0,Y 201.236,Z 723.359,A -85,B 0,C 180,E1 -22018.996,E2 -22018.996} C_VEL
LIN {X 0,Y 198.088,Z 733.769,A -85,B 0,C 180,E1 -22021.094,E2 -22021.094} C_VEL
LIN {X 0,Y 195.168,Z 742.283,A -85,B 0,C 180,E1 -22023.251,E2 -22023.251} C_VEL
LIN {X 0,Y 192.441,Z 750.144,A -85,B 0,C 180,E1 -22025.744,E2 -22025.744} C_VEL
LIN {X 0,Y 189.604,Z 757.825,A -85,B 0,C 180,E1 -22028.816,E2 -22028.816} C_VEL
LIN {X 0,Y 186.857,Z 764.909,A -85,B 0,C 180,E1 -22032.491,E2 -22032.491} C_VEL
LIN {X 0,Y 185.124,Z 769.626,A -85,B 0,C 180,E1 -22035.716,E2 -22035.716} C_VEL
LIN {X 0,Y 183.993,Z 773.239,A -85,B 0,C 180,E1 -22038.992,E2 -22038.992} C_VEL
LIN {X 0,Y 183.507,Z 775.103,A -85,B 0,C 180,E1 -22041.19,E2 -22041.19} C_VEL
LIN {X 0,Y 183.211,Z 776.5,A -85,B 0,C 180,E1 -22043.394,E2 -22043.394} C_VEL
LIN {X 0,Y 183.05,Z 778.108,A -85,B 0,C 180,E1 -22047.802,E2 -22047.802} C_VEL
LIN {X 0,Y 183.143,Z 778.322,A -85,B 0,C 180,E1 -22050.002,E2 -22050.002} C_VEL
LIN {X 0,Y 183.207,Z 778.098,A -85,B 0,C 180,E1 -22052.2,E2 -22052.2} C_VEL
LIN {X 0,Y 183.867,Z 776.494,A -85,B 0,C 180,E1 -22056.587,E2 -22056.587} C_VEL
LIN {X 0,Y 183.973,Z 776.596,A -85,B 0,C 180,E1 -22057.134,E2 -22057.134} C_VEL
LIN {X 0,Y 184.687,Z 780.16,A -85,B 0,C 180,E1 -22060.97,E2 -22060.97} C_VEL
LIN {X 0,Y 185.625,Z 781.59,A -85,B 0,C 180,E1 -22063.132,E2 -22063.132} C_VEL
LIN {X 0,Y 186.865,Z 782.474,A -85,B 0,C 180,E1 -22065.266,E2 -22065.266} C_VEL
LIN {X 0,Y 188.36,Z 782.84,A -85,B 0,C 180,E1 -22067.369,E2 -22067.369} C_VEL
LIN {X 0,Y 190.17,Z 782.782,A -85,B 0,C 180,E1 -22069.429,E2 -22069.429} C_VEL
LIN {X 0,Y 192.332,Z 782.288,A -85,B 0,C 180,E1 -22071.435,E2 -22071.435} C_VEL
LIN {X 0,Y 194.994,Z 781.298,A -85,B 0,C 180,E1 -22073.359,E2 -22073.359} C_VEL
LIN {X 0,Y 199.282,Z 778.833,A -85,B 0,C 180,E1 -22076.159,E2 -22076.159} C_VEL
LIN {X 0,Y 204.248,Z 775.18,A -85,B 0,C 180,E1 -22078.8,E2 -22078.8} C_VEL
LIN {X 0,Y 209.714,Z 770.278,A -85,B 0,C 180,E1 -22081.297,E2 -22081.297} C_VEL
LIN {X 0,Y 215.726,Z 763.926,A -85,B 0,C 180,E1 -22083.632,E2 -22083.632} C_VEL
LIN {X 0,Y 221.076,Z 757.191,A -85,B 0,C 180,E1 -22085.464,E2 -22085.464} C_VEL
LIN {X 0,Y 226.87,Z 748.968,A -85,B 0,C 180,E1 -22087.164,E2 -22087.164} C_VEL
LIN {X 0,Y 232.255,Z 739.688,A -85,B 0,C 180,E1 -22088.618,E2 -22088.618} C_VEL
LIN {X 0,Y 237.858,Z 728.125,A -85,B 0,C 180,E1 -22089.991,E2 -22089.991} C_VEL
LIN {X 0,Y 241.697,Z 718.047,A -85,B 0,C 180,E1 -22090.865,E2 -22090.865} C_VEL
LIN {X 0,Y 245.334,Z 705.593,A -85,B 0,C 180,E1 -22091.695,E2 -22091.695} C_VEL
LIN {X 0,Y 253.821,Z 671.722,A -85,B 0,C 180,E1 -22093.457,E2 -22093.457} C_VEL
LIN {X 0,Y 254.9,Z 667.417,A -85,B 0,C 180,E1 -22093.697,E2 -22093.697} C_VEL
LIN {X 0,Y 254.342,Z 669.251,A -85,B 0,C 180,E1 -22095.858,E2 -22095.858} C_VEL
LIN {X 0,Y 254.231,Z 669.818,A -85,B 0,C 180,E1 -22096.226,E2 -22096.226} C_VEL
LIN {X 0,Y 251.921,Z 681.568,A -85,B 0,C 180,E1 -22098.375,E2 -22098.375} C_VEL
LIN {X 0,Y 250.8,Z 688.228,A -85,B 0,C 180,E1 -22099.38,E2 -22099.38} C_VEL
LIN {X 0,Y 245.264,Z 711.031,A -85,B 0,C 180,E1 -22100.522,E2 -22100.522} C_VEL
LIN {X 0,Y 241.581,Z 722.273,A -85,B 0,C 180,E1 -22101.283,E2 -22101.283} C_VEL
LIN {X 0,Y 237.608,Z 731.79,A -85,B 0,C 180,E1 -22102.139,E2 -22102.139} C_VEL
LIN {X 0,Y 233.124,Z 740.755,A -85,B 0,C 180,E1 -22103.189,E2 -22103.189} C_VEL
LIN {X 0,Y 227.619,Z 749.765,A -85,B 0,C 180,E1 -22104.625,E2 -22104.625} C_VEL
LIN {X 0,Y 222.927,Z 756.446,A -85,B 0,C 180,E1 -22105.973,E2 -22105.973} C_VEL
LIN {X 0,Y 217.493,Z 763.118,A -85,B 0,C 180,E1 -22107.713,E2 -22107.713} C_VEL
LIN {X 0,Y 211.136,Z 769.578,A -85,B 0,C 180,E1 -22110.046,E2 -22110.046} C_VEL
LIN {X 0,Y 205.49,Z 774.36,A -85,B 0,C 180,E1 -22112.502,E2 -22112.502} C_VEL
LIN {X 0,Y 200.347,Z 777.807,A -85,B 0,C 180,E1 -22115.105,E2 -22115.105} C_VEL
LIN {X 0,Y 197.22,Z 779.377,A -85,B 0,C 180,E1 -22116.922,E2 -22116.922} C_VEL
LIN {X 0,Y 194.38,Z 780.389,A -85,B 0,C 180,E1 -22118.804,E2 -22118.804} C_VEL
LIN {X 0,Y 191.9,Z 780.916,A -85,B 0,C 180,E1 -22120.755,E2 -22120.755} C_VEL
LIN {X 0,Y 189.801,Z 780.979,A -85,B 0,C 180,E1 -22122.769,E2 -22122.769} C_VEL
LIN {X 0,Y 188.043,Z 780.57,A -85,B 0,C 180,E1 -22124.834,E2 -22124.834} C_VEL
LIN {X 0,Y 186.592,Z 779.621,A -85,B 0,C 180,E1 -22126.939,E2 -22126.939} C_VEL
LIN {X 0,Y 185.459,Z 778.144,A -85,B 0,C 180,E1 -22129.078,E2 -22129.078} C_VEL
LIN {X 0,Y 184.277,Z 774.771,A -85,B 0,C 180,E1 -22132.578,E2 -22132.578} C_VEL
LIN {X 0,Y 183.994,Z 770.649,A -85,B 0,C 180,E1 -22135.619,E2 -22135.619} C_VEL
LIN {X 0,Y 184.124,Z 764.681,A -85,B 0,C 180,E1 -22138.907,E2 -22138.907} C_VEL
LIN {X 0,Y 184.445,Z 758.356,A -85,B 0,C 180,E1 -22141.638,E2 -22141.638} C_VEL
LIN {X 0,Y 184.756,Z 750.125,A -85,B 0,C 180,E1 -22144.363,E2 -22144.363} C_VEL
LIN {X 0,Y 185.131,Z 743.032,A -85,B 0,C 180,E1 -22146.266,E2 -22146.266} C_VEL
LIN {X 0,Y 185.507,Z 732.773,A -85,B 0,C 180,E1 -22148.442,E2 -22148.442} C_VEL
LIN {X 0,Y 186.026,Z 722.928,A -85,B 0,C 180,E1 -22150.052,E2 -22150.052} C_VEL
LIN {X 0,Y 186.398,Z 711.232,A -85,B 0,C 180,E1 -22151.485,E2 -22151.485} C_VEL
LIN {X 0,Y 186.793,Z 699.055,A -85,B 0,C 180,E1 -22152.515,E2 -22152.515} C_VEL
LIN {X 0,Y 187.395,Z 656.724,A -85,B 0,C 180,E1 -22155.534,E2 -22155.534} C_VEL
LIN {X 0,Y 186.086,Z 634.642,A -85,B 0,C 180,E1 -22157.02,E2 -22157.02} C_VEL
LIN {X 0,Y 186.046,Z 632.282,A -85,B 0,C 180,E1 -22157.236,E2 -22157.236} C_VEL
LIN {X 0,Y 188.014,Z 609.445,A -85,B 0,C 180,E1 -22163.693,E2 -22163.693} C_VEL
LIN {X 0,Y 190.28,Z 589.432,A -85,B 0,C 180,E1 -22169.301,E2 -22169.301} C_VEL
LIN {X 0,Y 190.577,Z 585.249,A -85,B 0,C 180,E1 -22170.469,E2 -22170.469} C_VEL
LIN {X 0,Y 186.97,Z 567.842,A -85,B 0,C 180,E1 -22175.622,E2 -22175.622} C_VEL
LIN {X 0,Y 185.691,Z 561.538,A -85,B 0,C 180,E1 -22177.623,E2 -22177.623} C_VEL
LIN {X 0,Y 185.486,Z 561.504,A -85,B 0,C 180,E1 -22182.225,E2 -22182.225} C_VEL
LIN {X 0,Y 185.723,Z 562.445,A -85,B 0,C 180,E1 -22182.778,E2 -22182.778} C_VEL
LIN {X 0,Y 187.333,Z 565.301,A -85,B 0,C 180,E1 -22183.51,E2 -22183.51} C_VEL
LIN {X 0,Y 188.864,Z 566.866,A -85,B 0,C 180,E1 -22184.085,E2 -22184.085} C_VEL
LIN {X 0,Y 191.113,Z 570.291,A -85,B 0,C 180,E1 -22184.961,E2 -22184.961} C_VEL
LIN {X 0,Y 192.918,Z 572.964,A -85,B 0,C 180,E1 -22185.637,E2 -22185.637} C_VEL
LIN {X 0,Y 197.474,Z 579.596,A -85,B 0,C 180,E1 -22187.249,E2 -22187.249} C_VEL
LIN {X 0,Y 204.225,Z 590.92,A -85,B 0,C 180,E1 -22189.507,E2 -22189.507} C_VEL
LIN {X 0,Y 210.887,Z 605.401,A -85,B 0,C 180,E1 -22191.667,E2 -22191.667} C_VEL
LIN {X 0,Y 213.474,Z 611.904,A -85,B 0,C 180,E1 -22192.49,E2 -22192.49} C_VEL
LIN {X 0,Y 210.854,Z 663.922,A -85,B 0,C 180,E1 -22194.167,E2 -22194.167} C_VEL
LIN {X 0,Y 209.431,Z 676.992,A -85,B 0,C 180,E1 -22194.898,E2 -22194.898} C_VEL
LIN {X 0,Y 207.511,Z 689.953,A -85,B 0,C 180,E1 -22196.024,E2 -22196.024} C_VEL
LIN {X 0,Y 205.288,Z 701.236,A -85,B 0,C 180,E1 -22197.369,E2 -22197.369} C_VEL
LIN {X 0,Y 202.265,Z 712.867,A -85,B 0,C 180,E1 -22199.167,E2 -22199.167} C_VEL
LIN {X 0,Y 199.196,Z 723.312,A -85,B 0,C 180,E1 -22201.266,E2 -22201.266} C_VEL
LIN {X 0,Y 196.307,Z 732.432,A -85,B 0,C 180,E1 -22203.606,E2 -22203.606} C_VEL
LIN {X 0,Y 193.262,Z 741.079,A -85,B 0,C 180,E1 -22206.419,E2 -22206.419} C_VEL
LIN {X 0,Y 190.355,Z 748.482,A -85,B 0,C 180,E1 -22209.465,E2 -22209.465} C_VEL
LIN {X 0,Y 188.034,Z 754.421,A -85,B 0,C 180,E1 -22212.6,E2 -22212.6} C_VEL
LIN {X 0,Y 186.129,Z 759.112,A -85,B 0,C 180,E1 -22215.791,E2 -22215.791} C_VEL
LIN {X 0,Y 184.759,Z 762.695,A -85,B 0,C 180,E1 -22219.034,E2 -22219.034} C_VEL
LIN {X 0,Y 184.117,Z 764.544,A -85,B 0,C 180,E1 -22221.215,E2 -22221.215} C_VEL
LIN {X 0,Y 183.459,Z 766.665,A -85,B 0,C 180,E1 -22224.888,E2 -22224.888} C_VEL
LIN {X 0,Y 183.229,Z 767.53,A -85,B 0,C 180,E1 -22227.8,E2 -22227.8} C_VEL
LIN {X 0,Y 183.212,Z 767.757,A -85,B 0,C 180,E1 -22229.998,E2 -22229.998} C_VEL
LIN {X 0,Y 183.228,Z 767.564,A -85,B 0,C 180,E1 -22232.196,E2 -22232.196} C_VEL
LIN {X 0,Y 183.458,Z 766.722,A -85,B 0,C 180,E1 -22235.111,E2 -22235.111} C_VEL
LIN {X 0,Y 184.114,Z 764.659,A -85,B 0,C 180,E1 -22238.781,E2 -22238.781} C_VEL
LIN {X 0,Y 185.129,Z 761.79,A -85,B 0,C 180,E1 -22242.05,E2 -22242.05} C_VEL
LIN {X 0,Y 186.66,Z 757.895,A -85,B 0,C 180,E1 -22245.279,E2 -22245.279} C_VEL
LIN {X 0,Y 188.68,Z 752.875,A -85,B 0,C 180,E1 -22248.456,E2 -22248.456} C_VEL
LIN {X 0,Y 191.201,Z 746.548,A -85,B 0,C 180,E1 -22251.564,E2 -22251.564} C_VEL
LIN {X 0,Y 194.283,Z 738.627,A -85,B 0,C 180,E1 -22254.58,E2 -22254.58} C_VEL
LIN {X 0,Y 196.996,Z 730.617,A -85,B 0,C 180,E1 -22257.035,E2 -22257.035} C_VEL
LIN {X 0,Y 200.12,Z 720.703,A -85,B 0,C 180,E1 -22259.448,E2 -22259.448} C_VEL
LIN {X 0,Y 203.271,Z 709.605,A -85,B 0,C 180,E1 -22261.527,E2 -22261.527} C_VEL
LIN {X 0,Y 205.864,Z 698.719,A -85,B 0,C 180,E1 -22263.106,E2 -22263.106} C_VEL
LIN {X 0,Y 208.162,Z 686.677,A -85,B 0,C 180,E1 -22264.436,E2 -22264.436} C_VEL
LIN {X 0,Y 209.98,Z 674.139,A -85,B 0,C 180,E1 -22265.42,E2 -22265.42} C_VEL
LIN {X 0,Y 211.146,Z 661.567,A -85,B 0,C 180,E1 -22266.054,E2 -22266.054} C_VEL
LIN {X 0,Y 213.608,Z 611.991,A -85,B 0,C 180,E1 -22267.637,E2 -22267.637} C_VEL
LIN {X 0,Y 207.306,Z 597.323,A -85,B 0,C 180,E1 -22269.647,E2 -22269.647} C_VEL
LIN {X 0,Y 202.764,Z 588.173,A -85,B 0,C 180,E1 -22271.147,E2 -22271.147} C_VEL
LIN {X 0,Y 196.137,Z 577.725,A -85,B 0,C 180,E1 -22273.388,E2 -22273.388} C_VEL
LIN {X 0,Y 193.147,Z 573.365,A -85,B 0,C 180,E1 -22274.46,E2 -22274.46} C_VEL
LIN {X 0,Y 190.906,Z 570.061,A -85,B 0,C 180,E1 -22275.302,E2 -22275.302} C_VEL
LIN {X 0,Y 188.765,Z 566.69,A -85,B 0,C 180,E1 -22276.148,E2 -22276.148} C_VEL
LIN {X 0,Y 186.39,Z 564.057,A -85,B 0,C 180,E1 -22277.064,E2 -22277.064} C_VEL
LIN {X 0,Y 185.48,Z 561.378,A -85,B 0,C 180,E1 -22277.537,E2 -22277.537} C_VEL
LIN {X 0,Y 185.539,Z 561.34,A -85,B 0,C 180,E1 -22282.694,E2 -22282.694} C_VEL
LIN {X 0,Y 185.54,Z 561.363,A -85,B 0,C 180,E1 -22287.974,E2 -22287.974} C_VEL
LIN {X 0,Y 185.577,Z 561.366,A -85,B 0,C 180,E1 -22290.574,E2 -22290.574} C_VEL
LIN {X 0,Y 185.582,Z 561.367,A -85,B 0,C 180,E1 -22295.382,E2 -22295.382} C_VEL
LIN {X 0,Y 185.688,Z 561.354,A -85,B 0,C 180,E1 -22301.115,E2 -22301.115} C_VEL
LIN {X 0,Y 185.759,Z 561.345,A -85,B 0,C 180,E1 -22306.879,E2 -22306.879} C_VEL
LIN {X 0,Y 186.008,Z 561.297,A -85,B 0,C 180,E1 -22311.307,E2 -22311.307} C_VEL
LIN {X 0,Y 186.202,Z 561.271,A -85,B 0,C 180,E1 -22317.837,E2 -22317.837} C_VEL
LIN {X 0,Y 186.403,Z 561.267,A -85,B 0,C 180,E1 -22320,E2 -22320} C_VEL
LIN {X 0,Y 185.921,Z 561.306,A -85,B 0,C 180,E1 -22324.336,E2 -22324.336} C_VEL
LIN {X 0,Y 186.023,Z 561.3,A -85,B 0,C 180,E1 -22328.692,E2 -22328.692} C_VEL
LIN {X 0,Y 185.759,Z 561.346,A -85,B 0,C 180,E1 -22333.121,E2 -22333.121} C_VEL
LIN {X 0,Y 185.688,Z 561.355,A -85,B 0,C 180,E1 -22338.885,E2 -22338.885} C_VEL
LIN {X 0,Y 185.595,Z 561.367,A -85,B 0,C 180,E1 -22344.663,E2 -22344.663} C_VEL
LIN {X 0,Y 185.572,Z 561.368,A -85,B 0,C 180,E1 -22349.494,E2 -22349.494} C_VEL
LIN {X 0,Y 185.497,Z 561.358,A -85,B 0,C 180,E1 -22354.633,E2 -22354.633} C_VEL
LIN {X 0,Y 185.528,Z 561.369,A -85,B 0,C 180,E1 -22359.384,E2 -22359.384} C_VEL
LIN {X 0,Y 185.558,Z 561.614,A -85,B 0,C 180,E1 -22360.081,E2 -22360.081} C_VEL
LIN {X 0,Y 186.6,Z 565.145,A -85,B 0,C 180,E1 -22362.607,E2 -22362.607} C_VEL
LIN {X 0,Y 189.385,Z 569.763,A -85,B 0,C 180,E1 -22363.852,E2 -22363.852} C_VEL
LIN {X 0,Y 193.993,Z 577.447,A -85,B 0,C 180,E1 -22365.632,E2 -22365.632} C_VEL
LIN {X 0,Y 200.256,Z 588.795,A -85,B 0,C 180,E1 -22367.887,E2 -22367.887} C_VEL
LIN {X 0,Y 206.365,Z 601.888,A -85,B 0,C 180,E1 -22369.977,E2 -22369.977} C_VEL
LIN {X 0,Y 207.524,Z 605.34,A -85,B 0,C 180,E1 -22370.395,E2 -22370.395} C_VEL
LIN {X 0,Y 208.351,Z 611.009,A -85,B 0,C 180,E1 -22370.829,E2 -22370.829} C_VEL
LIN {X 0,Y 208.377,Z 616.92,A -85,B 0,C 180,E1 -22371.091,E2 -22371.091} C_VEL
LIN {X 0,Y 207.032,Z 633.308,A -85,B 0,C 180,E1 -22371.505,E2 -22371.505} C_VEL
LIN {X 0,Y 204.689,Z 674.929,A -85,B 0,C 180,E1 -22372.885,E2 -22372.885} C_VEL
LIN {X 0,Y 203.029,Z 688.811,A -85,B 0,C 180,E1 -22373.719,E2 -22373.719} C_VEL
LIN {X 0,Y 200.621,Z 701.515,A -85,B 0,C 180,E1 -22374.845,E2 -22374.845} C_VEL
LIN {X 0,Y 197.944,Z 713.186,A -85,B 0,C 180,E1 -22376.308,E2 -22376.308} C_VEL
LIN {X 0,Y 194.771,Z 724.45,A -85,B 0,C 180,E1 -22378.151,E2 -22378.151} C_VEL
LIN {X 0,Y 191.514,Z 734.6,A -85,B 0,C 180,E1 -22380.306,E2 -22380.306} C_VEL
LIN {X 0,Y 188.235,Z 743.75,A -85,B 0,C 180,E1 -22382.785,E2 -22382.785} C_VEL
LIN {X 0,Y 185.243,Z 751.874,A -85,B 0,C 180,E1 -22385.581,E2 -22385.581} C_VEL
LIN {X 0,Y 182.496,Z 758.742,A -85,B 0,C 180,E1 -22388.542,E2 -22388.542} C_VEL
LIN {X 0,Y 180.077,Z 764.706,A -85,B 0,C 180,E1 -22391.809,E2 -22391.809} C_VEL
LIN {X 0,Y 178.199,Z 769.421,A -85,B 0,C 180,E1 -22395.148,E2 -22395.148} C_VEL
LIN {X 0,Y 176.999,Z 773.035,A -85,B 0,C 180,E1 -22398.551,E2 -22398.551} C_VEL
LIN {X 0,Y 176.467,Z 774.898,A -85,B 0,C 180,E1 -22400.836,E2 -22400.836} C_VEL
LIN {X 0,Y 176.139,Z 776.295,A -85,B 0,C 180,E1 -22403.127,E2 -22403.127} C_VEL
LIN {X 0,Y 175.969,Z 777.904,A -85,B 0,C 180,E1 -22407.713,E2 -22407.713} C_VEL
LIN {X 0,Y 176.052,Z 778.117,A -85,B 0,C 180,E1 -22410.002,E2 -22410.002} C_VEL
LIN {X 0,Y 176.39,Z 777.28,A -85,B 0,C 180,E1 -22414.573,E2 -22414.573} C_VEL
LIN {X 0,Y 177.104,Z 775.811,A -85,B 0,C 180,E1 -22417.986,E2 -22417.986} C_VEL
LIN {X 0,Y 177.788,Z 779.155,A -85,B 0,C 180,E1 -22421.402,E2 -22421.402} C_VEL
LIN {X 0,Y 178.785,Z 780.742,A -85,B 0,C 180,E1 -22423.644,E2 -22423.644} C_VEL
LIN {X 0,Y 180.049,Z 781.883,A -85,B 0,C 180,E1 -22425.859,E2 -22425.859} C_VEL
LIN {X 0,Y 181.602,Z 782.6,A -85,B 0,C 180,E1 -22428.037,E2 -22428.037} C_VEL
LIN {X 0,Y 183.484,Z 782.842,A -85,B 0,C 180,E1 -22430.167,E2 -22430.167} C_VEL
LIN {X 0,Y 185.746,Z 782.555,A -85,B 0,C 180,E1 -22432.234,E2 -22432.234} C_VEL
LIN {X 0,Y 188.515,Z 781.82,A -85,B 0,C 180,E1 -22434.212,E2 -22434.212} C_VEL
LIN {X 0,Y 191.433,Z 780.657,A -85,B 0,C 180,E1 -22436.141,E2 -22436.141} C_VEL
LIN {X 0,Y 196.396,Z 777.942,A -85,B 0,C 180,E1 -22438.89,E2 -22438.89} C_VEL
LIN {X 0,Y 201.959,Z 774.063,A -85,B 0,C 180,E1 -22441.467,E2 -22441.467} C_VEL
LIN {X 0,Y 208.002,Z 768.935,A -85,B 0,C 180,E1 -22443.885,E2 -22443.885} C_VEL
LIN {X 0,Y 214.596,Z 762.143,A -85,B 0,C 180,E1 -22446.123,E2 -22446.123} C_VEL
LIN {X 0,Y 220.479,Z 755.147,A -85,B 0,C 180,E1 -22447.853,E2 -22447.853} C_VEL
LIN {X 0,Y 226.681,Z 746.396,A -85,B 0,C 180,E1 -22449.465,E2 -22449.465} C_VEL
LIN {X 0,Y 231.813,Z 737.857,A -85,B 0,C 180,E1 -22450.68,E2 -22450.68} C_VEL
LIN {X 0,Y 237.07,Z 727.253,A -85,B 0,C 180,E1 -22451.839,E2 -22451.839} C_VEL
LIN {X 0,Y 241.578,Z 715.961,A -85,B 0,C 180,E1 -22452.741,E2 -22452.741} C_VEL
LIN {X 0,Y 245.792,Z 701.43,A -85,B 0,C 180,E1 -22453.621,E2 -22453.621} C_VEL
LIN {X 0,Y 252.682,Z 675.314,A -85,B 0,C 180,E1 -22454.941,E2 -22454.941} C_VEL
LIN {X 0,Y 252.512,Z 676.008,A -85,B 0,C 180,E1 -22455.351,E2 -22455.351} C_VEL
LIN {X 0,Y 250.143,Z 686.303,A -85,B 0,C 180,E1 -22457.205,E2 -22457.205} C_VEL
LIN {X 0,Y 249.23,Z 690.707,A -85,B 0,C 180,E1 -22457.872,E2 -22457.872} C_VEL
LIN {X 0,Y 244.175,Z 710.415,A -85,B 0,C 180,E1 -22458.823,E2 -22458.823} C_VEL
LIN {X 0,Y 240.58,Z 721.346,A -85,B 0,C 180,E1 -22459.516,E2 -22459.516} C_VEL
LIN {X 0,Y 235.852,Z 732.106,A -85,B 0,C 180,E1 -22460.436,E2 -22460.436} C_VEL
LIN {X 0,Y 230.483,Z 742.054,A -85,B 0,C 180,E1 -22461.59,E2 -22461.59} C_VEL
LIN {X 0,Y 224.73,Z 750.864,A -85,B 0,C 180,E1 -22462.986,E2 -22462.986} C_VEL
LIN {X 0,Y 218.592,Z 758.81,A -85,B 0,C 180,E1 -22464.639,E2 -22464.639} C_VEL
LIN {X 0,Y 211.605,Z 766.171,A -85,B 0,C 180,E1 -22466.769,E2 -22466.769} C_VEL
LIN {X 0,Y 207.28,Z 770.101,A -85,B 0,C 180,E1 -22468.295,E2 -22468.295} C_VEL
LIN {X 0,Y 201.26,Z 774.745,A -85,B 0,C 180,E1 -22470.733,E2 -22470.733} C_VEL
LIN {X 0,Y 197.511,Z 777.069,A -85,B 0,C 180,E1 -22472.447,E2 -22472.447} C_VEL
LIN {X 0,Y 193.982,Z 778.84,A -85,B 0,C 180,E1 -22474.23,E2 -22474.23} C_VEL
LIN {X 0,Y 190.742,Z 780.098,A -85,B 0,C 180,E1 -22476.09,E2 -22476.09} C_VEL
LIN {X 0,Y 187.798,Z 780.89,A -85,B 0,C 180,E1 -22478.023,E2 -22478.023} C_VEL
LIN {X 0,Y 185.218,Z 781.15,A -85,B 0,C 180,E1 -22480.032,E2 -22480.032} C_VEL
LIN {X 0,Y 183.046,Z 780.865,A -85,B 0,C 180,E1 -22482.112,E2 -22482.112} C_VEL
LIN {X 0,Y 181.226,Z 780.128,A -85,B 0,C 180,E1 -22484.249,E2 -22484.249} C_VEL
LIN {X 0,Y 179.732,Z 778.938,A -85,B 0,C 180,E1 -22486.431,E2 -22486.431} C_VEL
LIN {X 0,Y 178.125,Z 776.201,A -85,B 0,C 180,E1 -22489.773,E2 -22489.773} C_VEL
LIN {X 0,Y 177.22,Z 772.271,A -85,B 0,C 180,E1 -22493.167,E2 -22493.167} C_VEL
LIN {X 0,Y 177.142,Z 767.009,A -85,B 0,C 180,E1 -22496.588,E2 -22496.588} C_VEL
LIN {X 0,Y 177.353,Z 761.294,A -85,B 0,C 180,E1 -22499.432,E2 -22499.432} C_VEL
LIN {X 0,Y 177.708,Z 755.651,A -85,B 0,C 180,E1 -22501.7,E2 -22501.7} C_VEL
LIN {X 0,Y 177.912,Z 748.724,A -85,B 0,C 180,E1 -22503.964,E2 -22503.964} C_VEL
LIN {X 0,Y 178.297,Z 740.29,A -85,B 0,C 180,E1 -22506.223,E2 -22506.223} C_VEL
LIN {X 0,Y 178.66,Z 730.806,A -85,B 0,C 180,E1 -22508.198,E2 -22508.198} C_VEL
LIN {X 0,Y 179.156,Z 720.409,A -85,B 0,C 180,E1 -22509.921,E2 -22509.921} C_VEL
LIN {X 0,Y 179.516,Z 708.641,A -85,B 0,C 180,E1 -22511.289,E2 -22511.289} C_VEL
LIN {X 0,Y 179.863,Z 692.139,A -85,B 0,C 180,E1 -22512.624,E2 -22512.624} C_VEL
LIN {X 0,Y 180.352,Z 656.948,A -85,B 0,C 180,E1 -22515.25,E2 -22515.25} C_VEL
LIN {X 0,Y 179.013,Z 634.759,A -85,B 0,C 180,E1 -22516.831,E2 -22516.831} C_VEL
LIN {X 0,Y 178.963,Z 632.057,A -85,B 0,C 180,E1 -22517.13,E2 -22517.13} C_VEL
LIN {X 0,Y 181.036,Z 608.368,A -85,B 0,C 180,E1 -22524.056,E2 -22524.056} C_VEL
LIN {X 0,Y 183.53,Z 587.198,A -85,B 0,C 180,E1 -22530.173,E2 -22530.173} C_VEL
LIN {X 0,Y 182.459,Z 580.86,A -85,B 0,C 180,E1 -22532.067,E2 -22532.067} C_VEL
LIN {X 0,Y 178.684,Z 562.561,A -85,B 0,C 180,E1 -22537.763,E2 -22537.763} C_VEL
LIN {X 0,Y 178.508,Z 562.237,A -85,B 0,C 180,E1 -22539.045,E2 -22539.045} C_VEL
LIN {X 0,Y 178.559,Z 562.73,A -85,B 0,C 180,E1 -22540.037,E2 -22540.037} C_VEL
LIN {X 0,Y 179.073,Z 564.345,A -85,B 0,C 180,E1 -22540.564,E2 -22540.564} C_VEL
LIN {X 0,Y 180.957,Z 566.828,A -85,B 0,C 180,E1 -22541.411,E2 -22541.411} C_VEL
LIN {X 0,Y 182.016,Z 567.959,A -85,B 0,C 180,E1 -22541.857,E2 -22541.857} C_VEL
LIN {X 0,Y 184.219,Z 571.266,A -85,B 0,C 180,E1 -22542.809,E2 -22542.809} C_VEL
LIN {X 0,Y 185.441,Z 572.803,A -85,B 0,C 180,E1 -22543.303,E2 -22543.303} C_VEL
LIN {X 0,Y 191.904,Z 582.361,A -85,B 0,C 180,E1 -22545.822,E2 -22545.822} C_VEL
LIN {X 0,Y 198.964,Z 593.864,A -85,B 0,C 180,E1 -22548.33,E2 -22548.33} C_VEL
LIN {X 0,Y 205.258,Z 607.56,A -85,B 0,C 180,E1 -22550.5,E2 -22550.5} C_VEL
LIN {X 0,Y 207.781,Z 613.813,A -85,B 0,C 180,E1 -22551.348,E2 -22551.348} C_VEL
LIN {X 0,Y 205.147,Z 664.333,A -85,B 0,C 180,E1 -22553.021,E2 -22553.021} C_VEL
LIN {X 0,Y 203.657,Z 677.362,A -85,B 0,C 180,E1 -22553.763,E2 -22553.763} C_VEL
LIN {X 0,Y 201.681,Z 690.164,A -85,B 0,C 180,E1 -22554.9,E2 -22554.9} C_VEL
LIN {X 0,Y 199.353,Z 701.446,A -85,B 0,C 180,E1 -22556.27,E2 -22556.27} C_VEL
LIN {X 0,Y 196.224,Z 713.075,A -85,B 0,C 180,E1 -22558.108,E2 -22558.108} C_VEL
LIN {X 0,Y 193.012,Z 723.52,A -85,B 0,C 180,E1 -22560.255,E2 -22560.255} C_VEL
LIN {X 0,Y 189.827,Z 733.04,A -85,B 0,C 180,E1 -22562.773,E2 -22562.773} C_VEL
LIN {X 0,Y 186.775,Z 741.287,A -85,B 0,C 180,E1 -22565.547,E2 -22565.547} C_VEL
LIN {X 0,Y 183.726,Z 748.689,A -85,B 0,C 180,E1 -22568.689,E2 -22568.689} C_VEL
LIN {X 0,Y 181.251,Z 754.628,A -85,B 0,C 180,E1 -22571.927,E2 -22571.927} C_VEL
LIN {X 0,Y 179.242,Z 759.319,A -85,B 0,C 180,E1 -22575.233,E2 -22575.233} C_VEL
LIN {X 0,Y 177.792,Z 762.9,A -85,B 0,C 180,E1 -22578.599,E2 -22578.599} C_VEL
LIN {X 0,Y 177.096,Z 764.75,A -85,B 0,C 180,E1 -22580.864,E2 -22580.864} C_VEL
LIN {X 0,Y 176.358,Z 766.998,A -85,B 0,C 180,E1 -22585.053,E2 -22585.053} C_VEL
LIN {X 0,Y 176.145,Z 767.735,A -85,B 0,C 180,E1 -22587.711,E2 -22587.711} C_VEL
LIN {X 0,Y 176.121,Z 767.962,A -85,B 0,C 180,E1 -22589.998,E2 -22589.998} C_VEL
LIN {X 0,Y 176.144,Z 767.768,A -85,B 0,C 180,E1 -22592.285,E2 -22592.285} C_VEL
LIN {X 0,Y 176.364,Z 767.046,A -85,B 0,C 180,E1 -22594.968,E2 -22594.968} C_VEL
LIN {X 0,Y 177.094,Z 764.863,A -85,B 0,C 180,E1 -22599.132,E2 -22599.132} C_VEL
LIN {X 0,Y 178.186,Z 761.994,A -85,B 0,C 180,E1 -22602.527,E2 -22602.527} C_VEL
LIN {X 0,Y 179.803,Z 758.099,A -85,B 0,C 180,E1 -22605.877,E2 -22605.877} C_VEL
LIN {X 0,Y 181.936,Z 753.079,A -85,B 0,C 180,E1 -22609.166,E2 -22609.166} C_VEL
LIN {X 0,Y 184.619,Z 746.751,A -85,B 0,C 180,E1 -22612.373,E2 -22612.373} C_VEL
LIN {X 0,Y 187.845,Z 738.829,A -85,B 0,C 180,E1 -22615.482,E2 -22615.482} C_VEL
LIN {X 0,Y 190.95,Z 730.054,A -85,B 0,C 180,E1 -22618.222,E2 -22618.222} C_VEL
LIN {X 0,Y 194.289,Z 719.804,A -85,B 0,C 180,E1 -22620.724,E2 -22620.724} C_VEL
LIN {X 0,Y 197.635,Z 708.383,A -85,B 0,C 180,E1 -22622.838,E2 -22622.838} C_VEL
LIN {X 0,Y 200.376,Z 697.154,A -85,B 0,C 180,E1 -22624.439,E2 -22624.439} C_VEL
LIN {X 0,Y 202.751,Z 684.462,A -85,B 0,C 180,E1 -22625.796,E2 -22625.796} C_VEL
LIN {X 0,Y 204.659,Z 670.675,A -85,B 0,C 180,E1 -22626.794,E2 -22626.794} C_VEL
LIN {X 0,Y 205.679,Z 657.72,A -85,B 0,C 180,E1 -22627.372,E2 -22627.372} C_VEL
LIN {X 0,Y 207.941,Z 614.06,A -85,B 0,C 180,E1 -22628.769,E2 -22628.769} C_VEL
LIN {X 0,Y 201.329,Z 598.591,A -85,B 0,C 180,E1 -22631.022,E2 -22631.022} C_VEL
LIN {X 0,Y 197.811,Z 591.828,A -85,B 0,C 180,E1 -22632.245,E2 -22632.245} C_VEL
LIN {X 0,Y 191.845,Z 582.33,A -85,B 0,C 180,E1 -22634.382,E2 -22634.382} C_VEL
LIN {X 0,Y 186.906,Z 575.042,A -85,B 0,C 180,E1 -22636.29,E2 -22636.29} C_VEL
LIN {X 0,Y 184.509,Z 571.566,A -85,B 0,C 180,E1 -22637.274,E2 -22637.274} C_VEL
LIN {X 0,Y 182.16,Z 568.282,A -85,B 0,C 180,E1 -22638.277,E2 -22638.277} C_VEL
LIN {X 0,Y 181.392,Z 567.165,A -85,B 0,C 180,E1 -22638.617,E2 -22638.617} C_VEL
LIN {X 0,Y 179.418,Z 564.994,A -85,B 0,C 180,E1 -22639.473,E2 -22639.473} C_VEL
LIN {X 0,Y 178.492,Z 562.218,A -85,B 0,C 180,E1 -22640.037,E2 -22640.037} C_VEL
LIN {X 0,Y 178.492,Z 562.251,A -85,B 0,C 180,E1 -22645.773,E2 -22645.773} C_VEL
LIN {X 0,Y 178.518,Z 562.249,A -85,B 0,C 180,E1 -22650.005,E2 -22650.005} C_VEL
LIN {X 0,Y 178.529,Z 562.247,A -85,B 0,C 180,E1 -22654.874,E2 -22654.874} C_VEL
LIN {X 0,Y 178.633,Z 562.233,A -85,B 0,C 180,E1 -22660.769,E2 -22660.769} C_VEL
LIN {X 0,Y 178.676,Z 562.226,A -85,B 0,C 180,E1 -22666.349,E2 -22666.349} C_VEL
LIN {X 0,Y 178.957,Z 562.173,A -85,B 0,C 180,E1 -22670.962,E2 -22670.962} C_VEL
LIN {X 0,Y 179.148,Z 562.149,A -85,B 0,C 180,E1 -22677.752,E2 -22677.752} C_VEL
LIN {X 0,Y 179.366,Z 562.143,A -85,B 0,C 180,E1 -22680,E2 -22680} C_VEL
LIN {X 0,Y 178.869,Z 562.185,A -85,B 0,C 180,E1 -22684.507,E2 -22684.507} C_VEL
LIN {X 0,Y 178.972,Z 562.174,A -85,B 0,C 180,E1 -22689.037,E2 -22689.037} C_VEL
LIN {X 0,Y 178.677,Z 562.227,A -85,B 0,C 180,E1 -22693.651,E2 -22693.651} C_VEL
LIN {X 0,Y 178.632,Z 562.235,A -85,B 0,C 180,E1 -22699.231,E2 -22699.231} C_VEL
LIN {X 0,Y 178.528,Z 562.242,A -85,B 0,C 180,E1 -22705.125,E2 -22705.125} C_VEL
LIN {X 0,Y 178.471,Z 562.244,A -85,B 0,C 180,E1 -22710.792,E2 -22710.792} C_VEL
LIN {X 0,Y 178.481,Z 562.237,A -85,B 0,C 180,E1 -22714.221,E2 -22714.221} C_VEL
LIN {X 0,Y 178.527,Z 562.374,A -85,B 0,C 180,E1 -22718.067,E2 -22718.067} C_VEL
LIN {X 0,Y 179.289,Z 564.935,A -85,B 0,C 180,E1 -22720.025,E2 -22720.025} C_VEL
LIN {X 0,Y 181.779,Z 569.112,A -85,B 0,C 180,E1 -22721.275,E2 -22721.275} C_VEL
LIN {X 0,Y 186.529,Z 576.553,A -85,B 0,C 180,E1 -22723.311,E2 -22723.311} C_VEL
LIN {X 0,Y 191.843,Z 585.727,A -85,B 0,C 180,E1 -22725.431,E2 -22725.431} C_VEL
LIN {X 0,Y 197.413,Z 596.572,A -85,B 0,C 180,E1 -22727.518,E2 -22727.518} C_VEL
LIN {X 0,Y 203.975,Z 611.57,A -85,B 0,C 180,E1 -22729.852,E2 -22729.852} C_VEL
LIN {X 0,Y 206.532,Z 618.722,A -85,B 0,C 180,E1 -22730.758,E2 -22730.758} C_VEL
LIN {X 0,Y 207.315,Z 627.392,A -85,B 0,C 180,E1 -22731.311,E2 -22731.311} C_VEL
LIN {X 0,Y 207.032,Z 633.308,A -85,B 0,C 180,E1 -22731.505,E2 -22731.505} C_VEL
LIN {X 0,Y 206.228,Z 639.143,A -85,B 0,C 180,E1 -22731.582,E2 -22731.582} C_VEL
LIN {X 0,Y 200.778,Z 658.142,A -85,B 0,C 180,E1 -22731.203,E2 -22731.203} C_VEL
LIN {X 0,Y 199.861,Z 663.982,A -85,B 0,C 180,E1 -22731.256,E2 -22731.256} C_VEL
LIN {X 0,Y 198.766,Z 678.33,A -85,B 0,C 180,E1 -22731.837,E2 -22731.837} C_VEL
LIN {X 0,Y 196.995,Z 690.746,A -85,B 0,C 180,E1 -22732.666,E2 -22732.666} C_VEL
LIN {X 0,Y 194.64,Z 702.312,A -85,B 0,C 180,E1 -22733.756,E2 -22733.756} C_VEL
LIN {X 0,Y 191.673,Z 714.571,A -85,B 0,C 180,E1 -22735.368,E2 -22735.368} C_VEL
LIN {X 0,Y 188.378,Z 725.498,A -85,B 0,C 180,E1 -22737.253,E2 -22737.253} C_VEL
LIN {X 0,Y 184.641,Z 736.355,A -85,B 0,C 180,E1 -22739.715,E2 -22739.715} C_VEL
LIN {X 0,Y 181.288,Z 745.18,A -85,B 0,C 180,E1 -22742.279,E2 -22742.279} C_VEL
LIN {X 0,Y 177.965,Z 753.69,A -85,B 0,C 180,E1 -22745.456,E2 -22745.456} C_VEL
LIN {X 0,Y 174.937,Z 760.673,A -85,B 0,C 180,E1 -22748.806,E2 -22748.806} C_VEL
LIN {X 0,Y 172.585,Z 766.193,A -85,B 0,C 180,E1 -22752.219,E2 -22752.219} C_VEL
LIN {X 0,Y 170.829,Z 770.528,A -85,B 0,C 180,E1 -22755.711,E2 -22755.711} C_VEL
LIN {X 0,Y 170.026,Z 772.83,A -85,B 0,C 180,E1 -22758.075,E2 -22758.075} C_VEL
LIN {X 0,Y 169.424,Z 774.692,A -85,B 0,C 180,E1 -22760.451,E2 -22760.451} C_VEL
LIN {X 0,Y 169.073,Z 776.09,A -85,B 0,C 180,E1 -22762.839,E2 -22762.839} C_VEL
LIN {X 0,Y 168.862,Z 777.699,A -85,B 0,C 180,E1 -22767.617,E2 -22767.617} C_VEL
LIN {X 0,Y 168.963,Z 777.913,A -85,B 0,C 180,E1 -22770.002,E2 -22770.002} C_VEL
LIN {X 0,Y 169.326,Z 777.076,A -85,B 0,C 180,E1 -22774.764,E2 -22774.764} C_VEL
LIN {X 0,Y 170.331,Z 775.14,A -85,B 0,C 180,E1 -22779.128,E2 -22779.128} C_VEL
LIN {X 0,Y 170.969,Z 777.864,A -85,B 0,C 180,E1 -22781.863,E2 -22781.863} C_VEL
LIN {X 0,Y 171.958,Z 779.799,A -85,B 0,C 180,E1 -22784.197,E2 -22784.197} C_VEL
LIN {X 0,Y 173.256,Z 781.241,A -85,B 0,C 180,E1 -22786.498,E2 -22786.498} C_VEL
LIN {X 0,Y 174.894,Z 782.128,A -85,B 0,C 180,E1 -22788.754,E2 -22788.754} C_VEL
LIN {X 0,Y 176.834,Z 782.604,A -85,B 0,C 180,E1 -22790.96,E2 -22790.96} C_VEL
LIN {X 0,Y 179.197,Z 782.684,A -85,B 0,C 180,E1 -22793.093,E2 -22793.093} C_VEL
LIN {X 0,Y 182.079,Z 782.309,A -85,B 0,C 180,E1 -22795.126,E2 -22795.126} C_VEL
LIN {X 0,Y 185.121,Z 781.4,A -85,B 0,C 180,E1 -22797.104,E2 -22797.104} C_VEL
LIN {X 0,Y 188.507,Z 780.022,A -85,B 0,C 180,E1 -22798.993,E2 -22798.993} C_VEL
LIN {X 0,Y 194.127,Z 777.119,A -85,B 0,C 180,E1 -22801.667,E2 -22801.667} C_VEL
LIN {X 0,Y 200.222,Z 773.029,A -85,B 0,C 180,E1 -22804.17,E2 -22804.17} C_VEL
LIN {X 0,Y 206.899,Z 767.543,A -85,B 0,C 180,E1 -22806.475,E2 -22806.475} C_VEL
LIN {X 0,Y 212.821,Z 761.764,A -85,B 0,C 180,E1 -22808.258,E2 -22808.258} C_VEL
LIN {X 0,Y 219.127,Z 754.788,A -85,B 0,C 180,E1 -22809.902,E2 -22809.902} C_VEL
LIN {X 0,Y 225.382,Z 746.402,A -85,B 0,C 180,E1 -22811.372,E2 -22811.372} C_VEL
LIN {X 0,Y 230.899,Z 737.809,A -85,B 0,C 180,E1 -22812.527,E2 -22812.527} C_VEL
LIN {X 0,Y 236.034,Z 728.219,A -85,B 0,C 180,E1 -22813.544,E2 -22813.544} C_VEL
LIN {X 0,Y 241.475,Z 715.19,A -85,B 0,C 180,E1 -22814.529,E2 -22814.529} C_VEL
LIN {X 0,Y 246.092,Z 699.911,A -85,B 0,C 180,E1 -22815.38,E2 -22815.38} C_VEL
LIN {X 0,Y 248.64,Z 690.57,A -85,B 0,C 180,E1 -22815.865,E2 -22815.865} C_VEL
LIN {X 0,Y 248.455,Z 691.329,A -85,B 0,C 180,E1 -22816.057,E2 -22816.057} C_VEL
LIN {X 0,Y 247.913,Z 693.463,A -85,B 0,C 180,E1 -22816.341,E2 -22816.341} C_VEL
LIN {X 0,Y 242.833,Z 712.347,A -85,B 0,C 180,E1 -22817.24,E2 -22817.24} C_VEL
LIN {X 0,Y 238.689,Z 723.541,A -85,B 0,C 180,E1 -22817.958,E2 -22817.958} C_VEL
LIN {X 0,Y 234.354,Z 732.703,A -85,B 0,C 180,E1 -22818.719,E2 -22818.719} C_VEL
LIN {X 0,Y 228.748,Z 742.561,A -85,B 0,C 180,E1 -22819.819,E2 -22819.819} C_VEL
LIN {X 0,Y 222.076,Z 752.099,A -85,B 0,C 180,E1 -22821.316,E2 -22821.316} C_VEL
LIN {X 0,Y 215.617,Z 759.734,A -85,B 0,C 180,E1 -22822.915,E2 -22822.915} C_VEL
LIN {X 0,Y 209.468,Z 765.834,A -85,B 0,C 180,E1 -22824.636,E2 -22824.636} C_VEL
LIN {X 0,Y 203.653,Z 770.698,A -85,B 0,C 180,E1 -22826.485,E2 -22826.485} C_VEL
LIN {X 0,Y 196.865,Z 775.469,A -85,B 0,C 180,E1 -22829.047,E2 -22829.047} C_VEL
LIN {X 0,Y 191.334,Z 778.347,A -85,B 0,C 180,E1 -22831.477,E2 -22831.477} C_VEL
LIN {X 0,Y 187.667,Z 779.832,A -85,B 0,C 180,E1 -22833.295,E2 -22833.295} C_VEL
LIN {X 0,Y 184.311,Z 780.745,A -85,B 0,C 180,E1 -22835.201,E2 -22835.201} C_VEL
LIN {X 0,Y 181.239,Z 781.142,A -85,B 0,C 180,E1 -22837.184,E2 -22837.184} C_VEL
LIN {X 0,Y 178.574,Z 781.09,A -85,B 0,C 180,E1 -22839.255,E2 -22839.255} C_VEL
LIN {X 0,Y 176.324,Z 780.599,A -85,B 0,C 180,E1 -22841.406,E2 -22841.406} C_VEL
LIN {X 0,Y 174.435,Z 779.632,A -85,B 0,C 180,E1 -22843.619,E2 -22843.619} C_VEL
LIN {X 0,Y 172.257,Z 777.229,A -85,B 0,C 180,E1 -22847.033,E2 -22847.033} C_VEL
LIN {X 0,Y 170.914,Z 773.662,A -85,B 0,C 180,E1 -22850.533,E2 -22850.533} C_VEL
LIN {X 0,Y 170.299,Z 768.904,A -85,B 0,C 180,E1 -22854.078,E2 -22854.078} C_VEL
LIN {X 0,Y 170.429,Z 762.647,A -85,B 0,C 180,E1 -22857.637,E2 -22857.637} C_VEL
LIN {X 0,Y 170.787,Z 755.891,A -85,B 0,C 180,E1 -22860.59,E2 -22860.59} C_VEL
LIN {X 0,Y 170.982,Z 751.024,A -85,B 0,C 180,E1 -22862.356,E2 -22862.356} C_VEL
LIN {X 0,Y 171.412,Z 742.035,A -85,B 0,C 180,E1 -22864.998,E2 -22864.998} C_VEL
LIN {X 0,Y 171.732,Z 733.161,A -85,B 0,C 180,E1 -22867.052,E2 -22867.052} C_VEL
LIN {X 0,Y 172.107,Z 723.464,A -85,B 0,C 180,E1 -22868.809,E2 -22868.809} C_VEL
LIN {X 0,Y 172.48,Z 713.181,A -85,B 0,C 180,E1 -22870.265,E2 -22870.265} C_VEL
LIN {X 0,Y 172.863,Z 699.655,A -85,B 0,C 180,E1 -22871.579,E2 -22871.579} C_VEL
LIN {X 0,Y 173.328,Z 657.204,A -85,B 0,C 180,E1 -22874.943,E2 -22874.943} C_VEL
LIN {X 0,Y 171.947,Z 634.34,A -85,B 0,C 180,E1 -22876.625,E2 -22876.625} C_VEL
LIN {X 0,Y 171.868,Z 631.962,A -85,B 0,C 180,E1 -22876.939,E2 -22876.939} C_VEL
LIN {X 0,Y 173.965,Z 608.185,A -85,B 0,C 180,E1 -22884.145,E2 -22884.145} C_VEL
LIN {X 0,Y 176.389,Z 587.915,A -85,B 0,C 180,E1 -22890.201,E2 -22890.201} C_VEL
LIN {X 0,Y 175.962,Z 584.365,A -85,B 0,C 180,E1 -22891.281,E2 -22891.281} C_VEL
LIN {X 0,Y 172.302,Z 566.84,A -85,B 0,C 180,E1 -22896.872,E2 -22896.872} C_VEL
LIN {X 0,Y 172.241,Z 565.927,A -85,B 0,C 180,E1 -22897.601,E2 -22897.601} C_VEL
LIN {X 0,Y 172.836,Z 566.418,A -85,B 0,C 180,E1 -22898.174,E2 -22898.174} C_VEL
LIN {X 0,Y 175.089,Z 568.736,A -85,B 0,C 180,E1 -22899.288,E2 -22899.288} C_VEL
LIN {X 0,Y 177.299,Z 572.154,A -85,B 0,C 180,E1 -22900.37,E2 -22900.37} C_VEL
LIN {X 0,Y 178.796,Z 573.936,A -85,B 0,C 180,E1 -22901.043,E2 -22901.043} C_VEL
LIN {X 0,Y 185.105,Z 583.042,A -85,B 0,C 180,E1 -22903.76,E2 -22903.76} C_VEL
LIN {X 0,Y 191.251,Z 592.718,A -85,B 0,C 180,E1 -22906.163,E2 -22906.163} C_VEL
LIN {X 0,Y 195.546,Z 600.448,A -85,B 0,C 180,E1 -22907.747,E2 -22907.747} C_VEL
LIN {X 0,Y 201.101,Z 613.109,A -85,B 0,C 180,E1 -22909.764,E2 -22909.764} C_VEL
LIN {X 0,Y 202.197,Z 615.871,A -85,B 0,C 180,E1 -22910.154,E2 -22910.154} C_VEL
LIN {X 0,Y 199.514,Z 664.827,A -85,B 0,C 180,E1 -22911.812,E2 -22911.812} C_VEL
LIN {X 0,Y 197.967,Z 677.734,A -85,B 0,C 180,E1 -22912.563,E2 -22912.563} C_VEL
LIN {X 0,Y 195.929,Z 690.376,A -85,B 0,C 180,E1 -22913.709,E2 -22913.709} C_VEL
LIN {X 0,Y 193.497,Z 701.656,A -85,B 0,C 180,E1 -22915.104,E2 -22915.104} C_VEL
LIN {X 0,Y 190.24,Z 713.284,A -85,B 0,C 180,E1 -22916.98,E2 -22916.98} C_VEL
LIN {X 0,Y 186.893,Z 723.728,A -85,B 0,C 180,E1 -22919.177,E2 -22919.177} C_VEL
LIN {X 0,Y 183.602,Z 733.041,A -85,B 0,C 180,E1 -22921.692,E2 -22921.692} C_VEL
LIN {X 0,Y 180.335,Z 741.494,A -85,B 0,C 180,E1 -22924.613,E2 -22924.613} C_VEL
LIN {X 0,Y 177.139,Z 748.895,A -85,B 0,C 180,E1 -22927.855,E2 -22927.855} C_VEL
LIN {X 0,Y 174.494,Z 754.835,A -85,B 0,C 180,E1 -22931.201,E2 -22931.201} C_VEL
LIN {X 0,Y 172.378,Z 759.525,A -85,B 0,C 180,E1 -22934.63,E2 -22934.63} C_VEL
LIN {X 0,Y 170.821,Z 763.106,A -85,B 0,C 180,E1 -22938.127,E2 -22938.127} C_VEL
LIN {X 0,Y 170.1,Z 764.955,A -85,B 0,C 180,E1 -22940.485,E2 -22940.485} C_VEL
LIN {X 0,Y 169.586,Z 766.343,A -85,B 0,C 180,E1 -22942.856,E2 -22942.856} C_VEL
LIN {X 0,Y 169.258,Z 767.332,A -85,B 0,C 180,E1 -22945.234,E2 -22945.234} C_VEL
LIN {X 0,Y 169.063,Z 767.939,A -85,B 0,C 180,E1 -22947.615,E2 -22947.615} C_VEL
LIN {X 0,Y 169.033,Z 768.166,A -85,B 0,C 180,E1 -22949.998,E2 -22949.998} C_VEL
LIN {X 0,Y 169.062,Z 767.973,A -85,B 0,C 180,E1 -22952.38,E2 -22952.38} C_VEL
LIN {X 0,Y 169.257,Z 767.388,A -85,B 0,C 180,E1 -22954.761,E2 -22954.761} C_VEL
LIN {X 0,Y 170.098,Z 765.067,A -85,B 0,C 180,E1 -22959.511,E2 -22959.511} C_VEL
LIN {X 0,Y 171.267,Z 762.197,A -85,B 0,C 180,E1 -22963.041,E2 -22963.041} C_VEL
LIN {X 0,Y 172.978,Z 758.303,A -85,B 0,C 180,E1 -22966.521,E2 -22966.521} C_VEL
LIN {X 0,Y 175.234,Z 753.282,A -85,B 0,C 180,E1 -22969.93,E2 -22969.93} C_VEL
LIN {X 0,Y 178.073,Z 746.953,A -85,B 0,C 180,E1 -22973.243,E2 -22973.243} C_VEL
LIN {X 0,Y 181.455,Z 739.031,A -85,B 0,C 180,E1 -22976.447,E2 -22976.447} C_VEL
LIN {X 0,Y 184.47,Z 730.925,A -85,B 0,C 180,E1 -22979.072,E2 -22979.072} C_VEL
LIN {X 0,Y 187.88,Z 721.106,A -85,B 0,C 180,E1 -22981.578,E2 -22981.578} C_VEL
LIN {X 0,Y 191.337,Z 710.005,A -85,B 0,C 180,E1 -22983.746,E2 -22983.746} C_VEL
LIN {X 0,Y 194.15,Z 699.116,A -85,B 0,C 180,E1 -22985.39,E2 -22985.39} C_VEL
LIN {X 0,Y 196.639,Z 687.07,A -85,B 0,C 180,E1 -22986.771,E2 -22986.771} C_VEL
LIN {X 0,Y 198.666,Z 674.061,A -85,B 0,C 180,E1 -22987.817,E2 -22987.817} C_VEL
LIN {X 0,Y 199.907,Z 661.058,A -85,B 0,C 180,E1 -22988.483,E2 -22988.483} C_VEL
LIN {X 0,Y 202.355,Z 616.194,A -85,B 0,C 180,E1 -22989.962,E2 -22989.962} C_VEL
LIN {X 0,Y 196.228,Z 601.687,A -85,B 0,C 180,E1 -22992.189,E2 -22992.189} C_VEL
LIN {X 0,Y 192.488,Z 594.74,A -85,B 0,C 180,E1 -22993.563,E2 -22993.563} C_VEL
LIN {X 0,Y 186.369,Z 584.944,A -85,B 0,C 180,E1 -22995.922,E2 -22995.922} C_VEL
LIN {X 0,Y 180.924,Z 577.001,A -85,B 0,C 180,E1 -22998.207,E2 -22998.207} C_VEL
LIN {X 0,Y 177.806,Z 572.682,A -85,B 0,C 180,E1 -22999.615,E2 -22999.615} C_VEL
LIN {X 0,Y 175.574,Z 569.645,A -85,B 0,C 180,E1 -23000.677,E2 -23000.677} C_VEL
LIN {X 0,Y 174.742,Z 568.282,A -85,B 0,C 180,E1 -23001.101,E2 -23001.101} C_VEL
LIN {X 0,Y 172.531,Z 566.133,A -85,B 0,C 180,E1 -23002.17,E2 -23002.17} C_VEL
LIN {X 0,Y 171.473,Z 563.587,A -85,B 0,C 180,E1 -23002.804,E2 -23002.804} C_VEL
LIN {X 0,Y 171.403,Z 563.102,A -85,B 0,C 180,E1 -23002.97,E2 -23002.97} C_VEL
LIN {X 0,Y 171.423,Z 563.12,A -85,B 0,C 180,E1 -23007.793,E2 -23007.793} C_VEL
LIN {X 0,Y 171.444,Z 563.125,A -85,B 0,C 180,E1 -23010.533,E2 -23010.533} C_VEL
LIN {X 0,Y 171.453,Z 563.123,A -85,B 0,C 180,E1 -23015.801,E2 -23015.801} C_VEL
LIN {X 0,Y 171.589,Z 563.111,A -85,B 0,C 180,E1 -23020.873,E2 -23020.873} C_VEL
LIN {X 0,Y 171.591,Z 563.102,A -85,B 0,C 180,E1 -23025.774,E2 -23025.774} C_VEL
LIN {X 0,Y 171.885,Z 563.052,A -85,B 0,C 180,E1 -23030.587,E2 -23030.587} C_VEL
LIN {X 0,Y 171.818,Z 563.068,A -85,B 0,C 180,E1 -23035.307,E2 -23035.307} C_VEL
LIN {X 0,Y 172.329,Z 563.02,A -85,B 0,C 180,E1 -23040,E2 -23040} C_VEL
LIN {X 0,Y 171.819,Z 563.064,A -85,B 0,C 180,E1 -23044.692,E2 -23044.692} C_VEL
LIN {X 0,Y 171.904,Z 563.052,A -85,B 0,C 180,E1 -23049.412,E2 -23049.412} C_VEL
LIN {X 0,Y 171.591,Z 563.104,A -85,B 0,C 180,E1 -23054.226,E2 -23054.226} C_VEL
LIN {X 0,Y 171.552,Z 563.114,A -85,B 0,C 180,E1 -23059.575,E2 -23059.575} C_VEL
LIN {X 0,Y 171.463,Z 563.118,A -85,B 0,C 180,E1 -23065.617,E2 -23065.617} C_VEL
LIN {X 0,Y 171.434,Z 563.121,A -85,B 0,C 180,E1 -23070.587,E2 -23070.587} C_VEL
LIN {X 0,Y 171.402,Z 563.184,A -85,B 0,C 180,E1 -23075.753,E2 -23075.753} C_VEL
LIN {X 0,Y 171.724,Z 564.407,A -85,B 0,C 180,E1 -23076.857,E2 -23076.857} C_VEL
LIN {X 0,Y 174.683,Z 569.116,A -85,B 0,C 180,E1 -23078.568,E2 -23078.568} C_VEL
LIN {X 0,Y 176.102,Z 571.144,A -85,B 0,C 180,E1 -23079.267,E2 -23079.267} C_VEL
LIN {X 0,Y 179.948,Z 577.16,A -85,B 0,C 180,E1 -23081.09,E2 -23081.09} C_VEL
LIN {X 0,Y 183.331,Z 582.762,A -85,B 0,C 180,E1 -23082.598,E2 -23082.598} C_VEL
LIN {X 0,Y 187.994,Z 591.096,A -85,B 0,C 180,E1 -23084.558,E2 -23084.558} C_VEL
LIN {X 0,Y 192.985,Z 600.998,A -85,B 0,C 180,E1 -23086.532,E2 -23086.532} C_VEL
LIN {X 0,Y 198.68,Z 614.324,A -85,B 0,C 180,E1 -23088.689,E2 -23088.689} C_VEL
LIN {X 0,Y 201.096,Z 620.645,A -85,B 0,C 180,E1 -23089.578,E2 -23089.578} C_VEL
LIN {X 0,Y 201.757,Z 628.427,A -85,B 0,C 180,E1 -23090.09,E2 -23090.09} C_VEL
LIN {X 0,Y 199.861,Z 663.982,A -85,B 0,C 180,E1 -23091.256,E2 -23091.256} C_VEL
LIN {X 0,Y 198.879,Z 669.809,A -85,B 0,C 180,E1 -23091.309,E2 -23091.309} C_VEL
LIN {X 0,Y 195.728,Z 679.212,A -85,B 0,C 180,E1 -23091.219,E2 -23091.219} C_VEL
LIN {X 0,Y 192.266,Z 688.514,A -85,B 0,C 180,E1 -23091.335,E2 -23091.335} C_VEL
LIN {X 0,Y 190.755,Z 694.084,A -85,B 0,C 180,E1 -23091.681,E2 -23091.681} C_VEL
LIN {X 0,Y 188.064,Z 705.997,A -85,B 0,C 180,E1 -23092.947,E2 -23092.947} C_VEL
LIN {X 0,Y 184.984,Z 717.317,A -85,B 0,C 180,E1 -23094.595,E2 -23094.595} C_VEL
LIN {X 0,Y 181.212,Z 728.824,A -85,B 0,C 180,E1 -23096.786,E2 -23096.786} C_VEL
LIN {X 0,Y 177.785,Z 738.096,A -85,B 0,C 180,E1 -23099.078,E2 -23099.078} C_VEL
LIN {X 0,Y 174.351,Z 746.554,A -85,B 0,C 180,E1 -23101.732,E2 -23101.732} C_VEL
LIN {X 0,Y 171.205,Z 754.129,A -85,B 0,C 180,E1 -23104.757,E2 -23104.757} C_VEL
LIN {X 0,Y 168.31,Z 760.469,A -85,B 0,C 180,E1 -23107.928,E2 -23107.928} C_VEL
LIN {X 0,Y 165.826,Z 765.989,A -85,B 0,C 180,E1 -23111.469,E2 -23111.469} C_VEL
LIN {X 0,Y 163.906,Z 770.323,A -85,B 0,C 180,E1 -23115.094,E2 -23115.094} C_VEL
LIN {X 0,Y 163.056,Z 772.625,A -85,B 0,C 180,E1 -23117.557,E2 -23117.557} C_VEL
LIN {X 0,Y 162.404,Z 774.488,A -85,B 0,C 180,E1 -23120.034,E2 -23120.034} C_VEL
LIN {X 0,Y 161.999,Z 775.885,A -85,B 0,C 180,E1 -23122.524,E2 -23122.524} C_VEL
LIN {X 0,Y 161.791,Z 776.884,A -85,B 0,C 180,E1 -23125.018,E2 -23125.018} C_VEL
LIN {X 0,Y 161.764,Z 777.548,A -85,B 0,C 180,E1 -23127.792,E2 -23127.792} C_VEL
LIN {X 0,Y 161.881,Z 777.709,A -85,B 0,C 180,E1 -23130.002,E2 -23130.002} C_VEL
LIN {X 0,Y 162.255,Z 776.871,A -85,B 0,C 180,E1 -23134.972,E2 -23134.972} C_VEL
LIN {X 0,Y 162.762,Z 775.867,A -85,B 0,C 180,E1 -23137.445,E2 -23137.445} C_VEL
LIN {X 0,Y 163.664,Z 774.416,A -85,B 0,C 180,E1 -23140.361,E2 -23140.361} C_VEL
LIN {X 0,Y 165.18,Z 778.608,A -85,B 0,C 180,E1 -23144.793,E2 -23144.793} C_VEL
LIN {X 0,Y 168.217,Z 781.5,A -85,B 0,C 180,E1 -23149.528,E2 -23149.528} C_VEL
LIN {X 0,Y 170.224,Z 782.307,A -85,B 0,C 180,E1 -23151.815,E2 -23151.815} C_VEL
LIN {X 0,Y 172.694,Z 782.598,A -85,B 0,C 180,E1 -23154.016,E2 -23154.016} C_VEL
LIN {X 0,Y 175.682,Z 782.477,A -85,B 0,C 180,E1 -23156.109,E2 -23156.109} C_VEL
LIN {X 0,Y 178.85,Z 781.948,A -85,B 0,C 180,E1 -23158.137,E2 -23158.137} C_VEL
LIN {X 0,Y 182.399,Z 780.978,A -85,B 0,C 180,E1 -23160.062,E2 -23160.062} C_VEL
LIN {X 0,Y 188.212,Z 778.541,A -85,B 0,C 180,E1 -23162.784,E2 -23162.784} C_VEL
LIN {X 0,Y 194.571,Z 775.008,A -85,B 0,C 180,E1 -23165.307,E2 -23165.307} C_VEL
LIN {X 0,Y 201.449,Z 770.234,A -85,B 0,C 180,E1 -23167.63,E2 -23167.63} C_VEL
LIN {X 0,Y 208.897,Z 764.106,A -85,B 0,C 180,E1 -23169.736,E2 -23169.736} C_VEL
LIN {X 0,Y 215.019,Z 757.96,A -85,B 0,C 180,E1 -23171.256,E2 -23171.256} C_VEL
LIN {X 0,Y 221.125,Z 750.984,A -85,B 0,C 180,E1 -23172.593,E2 -23172.593} C_VEL
LIN {X 0,Y 227.188,Z 742.826,A -85,B 0,C 180,E1 -23173.804,E2 -23173.804} C_VEL
LIN {X 0,Y 233.68,Z 732.261,A -85,B 0,C 180,E1 -23174.974,E2 -23174.974} C_VEL
LIN {X 0,Y 238.136,Z 723.43,A -85,B 0,C 180,E1 -23175.701,E2 -23175.701} C_VEL
LIN {X 0,Y 238.977,Z 721.628,A -85,B 0,C 180,E1 -23175.836,E2 -23175.836} C_VEL
LIN {X 0,Y 238.231,Z 723.313,A -85,B 0,C 180,E1 -23176.195,E2 -23176.195} C_VEL
LIN {X 0,Y 232.61,Z 734.697,A -85,B 0,C 180,E1 -23177.109,E2 -23177.109} C_VEL
LIN {X 0,Y 226.587,Z 744.299,A -85,B 0,C 180,E1 -23178.176,E2 -23178.176} C_VEL
LIN {X 0,Y 219.654,Z 753.467,A -85,B 0,C 180,E1 -23179.615,E2 -23179.615} C_VEL
LIN {X 0,Y 212.873,Z 760.824,A -85,B 0,C 180,E1 -23181.15,E2 -23181.15} C_VEL
LIN {X 0,Y 206.421,Z 766.689,A -85,B 0,C 180,E1 -23182.819,E2 -23182.819} C_VEL
LIN {X 0,Y 200.281,Z 771.445,A -85,B 0,C 180,E1 -23184.62,E2 -23184.62} C_VEL
LIN {X 0,Y 193.45,Z 775.737,A -85,B 0,C 180,E1 -23186.979,E2 -23186.979} C_VEL
LIN {X 0,Y 189.196,Z 777.869,A -85,B 0,C 180,E1 -23188.664,E2 -23188.664} C_VEL
LIN {X 0,Y 185.182,Z 779.443,A -85,B 0,C 180,E1 -23190.437,E2 -23190.437} C_VEL
LIN {X 0,Y 181.371,Z 780.52,A -85,B 0,C 180,E1 -23192.29,E2 -23192.29} C_VEL
LIN {X 0,Y 177.913,Z 781.132,A -85,B 0,C 180,E1 -23194.245,E2 -23194.245} C_VEL
LIN {X 0,Y 174.728,Z 781.303,A -85,B 0,C 180,E1 -23196.283,E2 -23196.283} C_VEL
LIN {X 0,Y 171.973,Z 780.953,A -85,B 0,C 180,E1 -23198.42,E2 -23198.42} C_VEL
LIN {X 0,Y 169.637,Z 780.104,A -85,B 0,C 180,E1 -23200.644,E2 -23200.644} C_VEL
LIN {X 0,Y 167.697,Z 778.82,A -85,B 0,C 180,E1 -23202.941,E2 -23202.941} C_VEL
LIN {X 0,Y 165.456,Z 776.032,A -85,B 0,C 180,E1 -23206.49,E2 -23206.49} C_VEL
LIN {X 0,Y 164.075,Z 772.14,A -85,B 0,C 180,E1 -23210.135,E2 -23210.135} C_VEL
LIN {X 0,Y 163.552,Z 765.871,A -85,B 0,C 180,E1 -23214.452,E2 -23214.452} C_VEL
LIN {X 0,Y 163.718,Z 760.134,A -85,B 0,C 180,E1 -23217.54,E2 -23217.54} C_VEL
LIN {X 0,Y 164.124,Z 752.921,A -85,B 0,C 180,E1 -23220.614,E2 -23220.614} C_VEL
LIN {X 0,Y 164.414,Z 744.498,A -85,B 0,C 180,E1 -23223.37,E2 -23223.37} C_VEL
LIN {X 0,Y 164.713,Z 737.712,A -85,B 0,C 180,E1 -23225.202,E2 -23225.202} C_VEL
LIN {X 0,Y 164.955,Z 729.392,A -85,B 0,C 180,E1 -23227.036,E2 -23227.036} C_VEL
LIN {X 0,Y 165.447,Z 718.837,A -85,B 0,C 180,E1 -23228.858,E2 -23228.858} C_VEL
LIN {X 0,Y 165.697,Z 707.86,A -85,B 0,C 180,E1 -23230.229,E2 -23230.229} C_VEL
LIN {X 0,Y 165.96,Z 690.77,A -85,B 0,C 180,E1 -23231.749,E2 -23231.749} C_VEL
LIN {X 0,Y 166.31,Z 656.927,A -85,B 0,C 180,E1 -23234.581,E2 -23234.581} C_VEL
LIN {X 0,Y 164.891,Z 633.609,A -85,B 0,C 180,E1 -23236.402,E2 -23236.402} C_VEL
LIN {X 0,Y 164.859,Z 632.315,A -85,B 0,C 180,E1 -23236.564,E2 -23236.564} C_VEL
LIN {X 0,Y 166.983,Z 606.882,A -85,B 0,C 180,E1 -23244.559,E2 -23244.559} C_VEL
LIN {X 0,Y 169.375,Z 587.498,A -85,B 0,C 180,E1 -23250.551,E2 -23250.551} C_VEL
LIN {X 0,Y 166.589,Z 574.399,A -85,B 0,C 180,E1 -23254.85,E2 -23254.85} C_VEL
LIN {X 0,Y 166.511,Z 573.635,A -85,B 0,C 180,E1 -23255.54,E2 -23255.54} C_VEL
LIN {X 0,Y 167.027,Z 574.063,A -85,B 0,C 180,E1 -23256.092,E2 -23256.092} C_VEL
LIN {X 0,Y 167.967,Z 574.543,A -85,B 0,C 180,E1 -23256.602,E2 -23256.602} C_VEL
LIN {X 0,Y 169.844,Z 574.183,A -85,B 0,C 180,E1 -23257.428,E2 -23257.428} C_VEL
LIN {X 0,Y 170.695,Z 573.649,A -85,B 0,C 180,E1 -23257.767,E2 -23257.767} C_VEL
LIN {X 0,Y 171.819,Z 574.41,A -85,B 0,C 180,E1 -23258.302,E2 -23258.302} C_VEL
LIN {X 0,Y 174.486,Z 578.31,A -85,B 0,C 180,E1 -23259.655,E2 -23259.655} C_VEL
LIN {X 0,Y 179.008,Z 584.775,A -85,B 0,C 180,E1 -23261.768,E2 -23261.768} C_VEL
LIN {X 0,Y 185.354,Z 594.509,A -85,B 0,C 180,E1 -23264.468,E2 -23264.468} C_VEL
LIN {X 0,Y 190.842,Z 604.238,A -85,B 0,C 180,E1 -23266.633,E2 -23266.633} C_VEL
LIN {X 0,Y 196.453,Z 617.285,A -85,B 0,C 180,E1 -23268.797,E2 -23268.797} C_VEL
LIN {X 0,Y 196.701,Z 617.958,A -85,B 0,C 180,E1 -23268.893,E2 -23268.893} C_VEL
LIN {X 0,Y 194.001,Z 664.7,A -85,B 0,C 180,E1 -23270.494,E2 -23270.494} C_VEL
LIN {X 0,Y 192.375,Z 678.11,A -85,B 0,C 180,E1 -23271.295,E2 -23271.295} C_VEL
LIN {X 0,Y 190.254,Z 690.588,A -85,B 0,C 180,E1 -23272.444,E2 -23272.444} C_VEL
LIN {X 0,Y 187.728,Z 701.865,A -85,B 0,C 180,E1 -23273.867,E2 -23273.867} C_VEL
LIN {X 0,Y 184.326,Z 713.493,A -85,B 0,C 180,E1 -23275.777,E2 -23275.777} C_VEL
LIN {X 0,Y 180.833,Z 723.936,A -85,B 0,C 180,E1 -23278.024,E2 -23278.024} C_VEL
LIN {X 0,Y 177.174,Z 733.767,A -85,B 0,C 180,E1 -23280.772,E2 -23280.772} C_VEL
LIN {X 0,Y 173.949,Z 741.7,A -85,B 0,C 180,E1 -23283.611,E2 -23283.611} C_VEL
LIN {X 0,Y 170.596,Z 749.101,A -85,B 0,C 180,E1 -23286.958,E2 -23286.958} C_VEL
LIN {X 0,Y 167.769,Z 755.041,A -85,B 0,C 180,E1 -23290.418,E2 -23290.418} C_VEL
LIN {X 0,Y 165.539,Z 759.731,A -85,B 0,C 180,E1 -23293.979,E2 -23293.979} C_VEL
LIN {X 0,Y 163.877,Z 763.312,A -85,B 0,C 180,E1 -23297.616,E2 -23297.616} C_VEL
LIN {X 0,Y 163.087,Z 765.161,A -85,B 0,C 180,E1 -23300.072,E2 -23300.072} C_VEL
LIN {X 0,Y 162.549,Z 766.548,A -85,B 0,C 180,E1 -23302.545,E2 -23302.545} C_VEL
LIN {X 0,Y 162.126,Z 767.715,A -85,B 0,C 180,E1 -23305.585,E2 -23305.585} C_VEL
LIN {X 0,Y 161.946,Z 768.371,A -85,B 0,C 180,E1 -23309.998,E2 -23309.998} C_VEL
LIN {X 0,Y 162.099,Z 767.81,A -85,B 0,C 180,E1 -23314.288,E2 -23314.288} C_VEL
LIN {X 0,Y 162.547,Z 766.627,A -85,B 0,C 180,E1 -23317.451,E2 -23317.451} C_VEL
LIN {X 0,Y 163.084,Z 765.271,A -85,B 0,C 180,E1 -23319.924,E2 -23319.924} C_VEL
LIN {X 0,Y 164.341,Z 762.402,A -85,B 0,C 180,E1 -23323.601,E2 -23323.601} C_VEL
LIN {X 0,Y 166.183,Z 758.507,A -85,B 0,C 180,E1 -23327.217,E2 -23327.217} C_VEL
LIN {X 0,Y 168.571,Z 753.486,A -85,B 0,C 180,E1 -23330.753,E2 -23330.753} C_VEL
LIN {X 0,Y 171.575,Z 747.156,A -85,B 0,C 180,E1 -23334.178,E2 -23334.178} C_VEL
LIN {X 0,Y 175.116,Z 739.234,A -85,B 0,C 180,E1 -23337.484,E2 -23337.484} C_VEL
LIN {X 0,Y 178.206,Z 731.341,A -85,B 0,C 180,E1 -23340.119,E2 -23340.119} C_VEL
LIN {X 0,Y 181.86,Z 721.307,A -85,B 0,C 180,E1 -23342.751,E2 -23342.751} C_VEL
LIN {X 0,Y 185.491,Z 710.204,A -85,B 0,C 180,E1 -23344.962,E2 -23344.962} C_VEL
LIN {X 0,Y 188.419,Z 699.315,A -85,B 0,C 180,E1 -23346.638,E2 -23346.638} C_VEL
LIN {X 0,Y 190.999,Z 687.267,A -85,B 0,C 180,E1 -23348.046,E2 -23348.046} C_VEL
LIN {X 0,Y 193.06,Z 674.74,A -85,B 0,C 180,E1 -23349.075,E2 -23349.075} C_VEL
LIN {X 0,Y 194.377,Z 661.787,A -85,B 0,C 180,E1 -23349.761,E2 -23349.761} C_VEL
LIN {X 0,Y 196.865,Z 618.295,A -85,B 0,C 180,E1 -23351.224,E2 -23351.224} C_VEL
LIN {X 0,Y 191.178,Z 604.754,A -85,B 0,C 180,E1 -23353.428,E2 -23353.428} C_VEL
LIN {X 0,Y 185.868,Z 595.301,A -85,B 0,C 180,E1 -23355.519,E2 -23355.519} C_VEL
LIN {X 0,Y 179.165,Z 585.01,A -85,B 0,C 180,E1 -23358.367,E2 -23358.367} C_VEL
LIN {X 0,Y 174.439,Z 578.211,A -85,B 0,C 180,E1 -23360.588,E2 -23360.588} C_VEL
LIN {X 0,Y 171.919,Z 574.52,A -85,B 0,C 180,E1 -23361.873,E2 -23361.873} C_VEL
LIN {X 0,Y 169.135,Z 571.336,A -85,B 0,C 180,E1 -23363.322,E2 -23363.322} C_VEL
LIN {X 0,Y 168.034,Z 569.36,A -85,B 0,C 180,E1 -23363.973,E2 -23363.973} C_VEL
LIN {X 0,Y 165.777,Z 567.468,A -85,B 0,C 180,E1 -23365.209,E2 -23365.209} C_VEL
LIN {X 0,Y 164.503,Z 564.906,A -85,B 0,C 180,E1 -23366.054,E2 -23366.054} C_VEL
LIN {X 0,Y 164.328,Z 564.01,A -85,B 0,C 180,E1 -23366.221,E2 -23366.221} C_VEL
LIN {X 0,Y 164.401,Z 564.002,A -85,B 0,C 180,E1 -23369.136,E2 -23369.136} C_VEL
LIN {X 0,Y 164.411,Z 564.005,A -85,B 0,C 180,E1 -23374.693,E2 -23374.693} C_VEL
LIN {X 0,Y 164.48,Z 563.992,A -85,B 0,C 180,E1 -23380.049,E2 -23380.049} C_VEL
LIN {X 0,Y 164.535,Z 563.974,A -85,B 0,C 180,E1 -23385.15,E2 -23385.15} C_VEL
LIN {X 0,Y 164.799,Z 563.933,A -85,B 0,C 180,E1 -23390.178,E2 -23390.178} C_VEL
LIN {X 0,Y 164.848,Z 563.946,A -85,B 0,C 180,E1 -23392.652,E2 -23392.652} C_VEL
LIN {X 0,Y 165.044,Z 563.904,A -85,B 0,C 180,E1 -23397.559,E2 -23397.559} C_VEL
LIN {X 0,Y 165.291,Z 563.896,A -85,B 0,C 180,E1 -23400,E2 -23400} C_VEL
LIN {X 0,Y 164.856,Z 563.949,A -85,B 0,C 180,E1 -23407.348,E2 -23407.348} C_VEL
LIN {X 0,Y 164.773,Z 563.942,A -85,B 0,C 180,E1 -23411.198,E2 -23411.198} C_VEL
LIN {X 0,Y 164.493,Z 563.981,A -85,B 0,C 180,E1 -23417.402,E2 -23417.402} C_VEL
LIN {X 0,Y 164.469,Z 563.992,A -85,B 0,C 180,E1 -23419.99,E2 -23419.99} C_VEL
LIN {X 0,Y 164.387,Z 563.996,A -85,B 0,C 180,E1 -23426.135,E2 -23426.135} C_VEL
LIN {X 0,Y 164.373,Z 564.005,A -85,B 0,C 180,E1 -23432.375,E2 -23432.375} C_VEL
LIN {X 0,Y 164.347,Z 564.225,A -85,B 0,C 180,E1 -23433.336,E2 -23433.336} C_VEL
LIN {X 0,Y 165.468,Z 567.045,A -85,B 0,C 180,E1 -23434.244,E2 -23434.244} C_VEL
LIN {X 0,Y 168.575,Z 570.289,A -85,B 0,C 180,E1 -23435.985,E2 -23435.985} C_VEL
LIN {X 0,Y 172.93,Z 576.961,A -85,B 0,C 180,E1 -23438.353,E2 -23438.353} C_VEL
LIN {X 0,Y 176.639,Z 582.907,A -85,B 0,C 180,E1 -23440.207,E2 -23440.207} C_VEL
LIN {X 0,Y 181.189,Z 590.599,A -85,B 0,C 180,E1 -23442.314,E2 -23442.314} C_VEL
LIN {X 0,Y 187.181,Z 602.279,A -85,B 0,C 180,E1 -23444.903,E2 -23444.903} C_VEL
LIN {X 0,Y 193.332,Z 616.597,A -85,B 0,C 180,E1 -23447.403,E2 -23447.403} C_VEL
LIN {X 0,Y 195.883,Z 623.34,A -85,B 0,C 180,E1 -23448.404,E2 -23448.404} C_VEL
LIN {X 0,Y 196.319,Z 629.046,A -85,B 0,C 180,E1 -23448.788,E2 -23448.788} C_VEL
LIN {X 0,Y 193.58,Z 674.357,A -85,B 0,C 180,E1 -23450.34,E2 -23450.34} C_VEL
LIN {X 0,Y 191.912,Z 687.614,A -85,B 0,C 180,E1 -23451.153,E2 -23451.153} C_VEL
LIN {X 0,Y 190.755,Z 694.084,A -85,B 0,C 180,E1 -23451.681,E2 -23451.681} C_VEL
LIN {X 0,Y 189.037,Z 699.617,A -85,B 0,C 180,E1 -23452.065,E2 -23452.065} C_VEL
LIN {X 0,Y 184.527,Z 708.351,A -85,B 0,C 180,E1 -23452.55,E2 -23452.55} C_VEL
LIN {X 0,Y 179.802,Z 716.713,A -85,B 0,C 180,E1 -23453.294,E2 -23453.294} C_VEL
LIN {X 0,Y 177.77,Z 721.65,A -85,B 0,C 180,E1 -23454.088,E2 -23454.088} C_VEL
LIN {X 0,Y 174.099,Z 731.889,A -85,B 0,C 180,E1 -23456.288,E2 -23456.288} C_VEL
LIN {X 0,Y 170.214,Z 741.473,A -85,B 0,C 180,E1 -23458.931,E2 -23458.931} C_VEL
LIN {X 0,Y 166.838,Z 749.33,A -85,B 0,C 180,E1 -23461.715,E2 -23461.715} C_VEL
LIN {X 0,Y 163.389,Z 757.011,A -85,B 0,C 180,E1 -23465.207,E2 -23465.207} C_VEL
LIN {X 0,Y 160.81,Z 762.273,A -85,B 0,C 180,E1 -23468.196,E2 -23468.196} C_VEL
LIN {X 0,Y 158.295,Z 767.372,A -85,B 0,C 180,E1 -23471.896,E2 -23471.896} C_VEL
LIN {X 0,Y 156.531,Z 771.344,A -85,B 0,C 180,E1 -23475.706,E2 -23475.706} C_VEL
LIN {X 0,Y 155.405,Z 774.283,A -85,B 0,C 180,E1 -23479.581,E2 -23479.581} C_VEL
LIN {X 0,Y 154.949,Z 775.68,A -85,B 0,C 180,E1 -23482.182,E2 -23482.182} C_VEL
LIN {X 0,Y 154.711,Z 776.679,A -85,B 0,C 180,E1 -23484.79,E2 -23484.79} C_VEL
LIN {X 0,Y 154.684,Z 777.404,A -85,B 0,C 180,E1 -23488.307,E2 -23488.307} C_VEL
LIN {X 0,Y 154.794,Z 777.504,A -85,B 0,C 180,E1 -23490.002,E2 -23490.002} C_VEL
LIN {X 0,Y 155.196,Z 776.666,A -85,B 0,C 180,E1 -23495.199,E2 -23495.199} C_VEL
LIN {X 0,Y 155.732,Z 775.664,A -85,B 0,C 180,E1 -23497.783,E2 -23497.783} C_VEL
LIN {X 0,Y 157.112,Z 773.576,A -85,B 0,C 180,E1 -23501.697,E2 -23501.697} C_VEL
LIN {X 0,Y 158.477,Z 777.231,A -85,B 0,C 180,E1 -23505.434,E2 -23505.434} C_VEL
LIN {X 0,Y 159.822,Z 779.209,A -85,B 0,C 180,E1 -23507.93,E2 -23507.93} C_VEL
LIN {X 0,Y 161.581,Z 780.644,A -85,B 0,C 180,E1 -23510.365,E2 -23510.365} C_VEL
LIN {X 0,Y 163.677,Z 781.667,A -85,B 0,C 180,E1 -23512.736,E2 -23512.736} C_VEL
LIN {X 0,Y 166.243,Z 782.335,A -85,B 0,C 180,E1 -23515.011,E2 -23515.011} C_VEL
LIN {X 0,Y 169.343,Z 782.57,A -85,B 0,C 180,E1 -23517.165,E2 -23517.165} C_VEL
LIN {X 0,Y 172.632,Z 782.283,A -85,B 0,C 180,E1 -23519.246,E2 -23519.246} C_VEL
LIN {X 0,Y 176.31,Z 781.585,A -85,B 0,C 180,E1 -23521.214,E2 -23521.214} C_VEL
LIN {X 0,Y 180.278,Z 780.486,A -85,B 0,C 180,E1 -23523.08,E2 -23523.08} C_VEL
LIN {X 0,Y 186.709,Z 777.887,A -85,B 0,C 180,E1 -23525.695,E2 -23525.695} C_VEL
LIN {X 0,Y 193.644,Z 774.204,A -85,B 0,C 180,E1 -23528.099,E2 -23528.099} C_VEL
LIN {X 0,Y 201.146,Z 769.285,A -85,B 0,C 180,E1 -23530.272,E2 -23530.272} C_VEL
LIN {X 0,Y 209.104,Z 762.83,A -85,B 0,C 180,E1 -23532.239,E2 -23532.239} C_VEL
LIN {X 0,Y 216.158,Z 755.975,A -85,B 0,C 180,E1 -23533.741,E2 -23533.741} C_VEL
LIN {X 0,Y 223.338,Z 747.837,A -85,B 0,C 180,E1 -23535.077,E2 -23535.077} C_VEL
LIN {X 0,Y 226.281,Z 743.916,A -85,B 0,C 180,E1 -23535.592,E2 -23535.592} C_VEL
LIN {X 0,Y 226.948,Z 743.061,A -85,B 0,C 180,E1 -23536.129,E2 -23536.129} C_VEL
LIN {X 0,Y 219.906,Z 752.163,A -85,B 0,C 180,E1 -23537.396,E2 -23537.396} C_VEL
LIN {X 0,Y 213.193,Z 759.43,A -85,B 0,C 180,E1 -23538.753,E2 -23538.753} C_VEL
LIN {X 0,Y 206.293,Z 765.539,A -85,B 0,C 180,E1 -23540.299,E2 -23540.299} C_VEL
LIN {X 0,Y 199.703,Z 770.508,A -85,B 0,C 180,E1 -23541.985,E2 -23541.985} C_VEL
LIN {X 0,Y 194.684,Z 773.679,A -85,B 0,C 180,E1 -23543.442,E2 -23543.442} C_VEL
LIN {X 0,Y 187.644,Z 777.332,A -85,B 0,C 180,E1 -23545.819,E2 -23545.819} C_VEL
LIN {X 0,Y 183.233,Z 779.067,A -85,B 0,C 180,E1 -23547.522,E2 -23547.522} C_VEL
LIN {X 0,Y 179.065,Z 780.319,A -85,B 0,C 180,E1 -23549.321,E2 -23549.321} C_VEL
LIN {X 0,Y 175.132,Z 781.131,A -85,B 0,C 180,E1 -23551.213,E2 -23551.213} C_VEL
LIN {X 0,Y 171.55,Z 781.4,A -85,B 0,C 180,E1 -23553.215,E2 -23553.215} C_VEL
LIN {X 0,Y 168.271,Z 781.166,A -85,B 0,C 180,E1 -23555.313,E2 -23555.313} C_VEL
LIN {X 0,Y 165.416,Z 780.512,A -85,B 0,C 180,E1 -23557.519,E2 -23557.519} C_VEL
LIN {X 0,Y 162.987,Z 779.446,A -85,B 0,C 180,E1 -23559.821,E2 -23559.821} C_VEL
LIN {X 0,Y 160.127,Z 776.932,A -85,B 0,C 180,E1 -23563.424,E2 -23563.424} C_VEL
LIN {X 0,Y 158.129,Z 773.315,A -85,B 0,C 180,E1 -23567.16,E2 -23567.16} C_VEL
LIN {X 0,Y 157.004,Z 768.391,A -85,B 0,C 180,E1 -23571.152,E2 -23571.152} C_VEL
LIN {X 0,Y 156.889,Z 762.435,A -85,B 0,C 180,E1 -23574.86,E2 -23574.86} C_VEL
LIN {X 0,Y 157.176,Z 755.923,A -85,B 0,C 180,E1 -23578.078,E2 -23578.078} C_VEL
LIN {X 0,Y 157.533,Z 749.537,A -85,B 0,C 180,E1 -23580.639,E2 -23580.639} C_VEL
LIN {X 0,Y 157.844,Z 740.446,A -85,B 0,C 180,E1 -23583.51,E2 -23583.51} C_VEL
LIN {X 0,Y 158.165,Z 731.324,A -85,B 0,C 180,E1 -23585.738,E2 -23585.738} C_VEL
LIN {X 0,Y 158.477,Z 721.515,A -85,B 0,C 180,E1 -23587.646,E2 -23587.646} C_VEL
LIN {X 0,Y 158.794,Z 710.558,A -85,B 0,C 180,E1 -23589.232,E2 -23589.232} C_VEL
LIN {X 0,Y 159.098,Z 696.648,A -85,B 0,C 180,E1 -23590.66,E2 -23590.66} C_VEL
LIN {X 0,Y 159.289,Z 656.622,A -85,B 0,C 180,E1 -23594.169,E2 -23594.169} C_VEL
LIN {X 0,Y 157.854,Z 632.573,A -85,B 0,C 180,E1 -23596.157,E2 -23596.157} C_VEL
LIN {X 0,Y 160.307,Z 603.442,A -85,B 0,C 180,E1 -23605.654,E2 -23605.654} C_VEL
LIN {X 0,Y 162.151,Z 587.418,A -85,B 0,C 180,E1 -23610.795,E2 -23610.795} C_VEL
LIN {X 0,Y 160.996,Z 582.162,A -85,B 0,C 180,E1 -23612.666,E2 -23612.666} C_VEL
LIN {X 0,Y 160.965,Z 581.571,A -85,B 0,C 180,E1 -23613.442,E2 -23613.442} C_VEL
LIN {X 0,Y 162.112,Z 582.408,A -85,B 0,C 180,E1 -23614.305,E2 -23614.305} C_VEL
LIN {X 0,Y 164.151,Z 582.051,A -85,B 0,C 180,E1 -23615.316,E2 -23615.316} C_VEL
LIN {X 0,Y 165.081,Z 581.413,A -85,B 0,C 180,E1 -23615.726,E2 -23615.726} C_VEL
LIN {X 0,Y 169.465,Z 581.497,A -85,B 0,C 180,E1 -23617.76,E2 -23617.76} C_VEL
LIN {X 0,Y 174.984,Z 589.323,A -85,B 0,C 180,E1 -23620.542,E2 -23620.542} C_VEL
LIN {X 0,Y 181.486,Z 599.566,A -85,B 0,C 180,E1 -23623.487,E2 -23623.487} C_VEL
LIN {X 0,Y 186.427,Z 608.52,A -85,B 0,C 180,E1 -23625.554,E2 -23625.554} C_VEL
LIN {X 0,Y 191.309,Z 620.112,A -85,B 0,C 180,E1 -23627.565,E2 -23627.565} C_VEL
LIN {X 0,Y 188.541,Z 665.513,A -85,B 0,C 180,E1 -23629.158,E2 -23629.158} C_VEL
LIN {X 0,Y 186.807,Z 678.932,A -85,B 0,C 180,E1 -23629.984,E2 -23629.984} C_VEL
LIN {X 0,Y 184.461,Z 691.879,A -85,B 0,C 180,E1 -23631.222,E2 -23631.222} C_VEL
LIN {X 0,Y 181.59,Z 703.656,A -85,B 0,C 180,E1 -23632.789,E2 -23632.789} C_VEL
LIN {X 0,Y 178.071,Z 714.991,A -85,B 0,C 180,E1 -23634.743,E2 -23634.743} C_VEL
LIN {X 0,Y 174.473,Z 725.199,A -85,B 0,C 180,E1 -23637.055,E2 -23637.055} C_VEL
LIN {X 0,Y 170.778,Z 734.52,A -85,B 0,C 180,E1 -23639.793,E2 -23639.793} C_VEL
LIN {X 0,Y 167.015,Z 743.254,A -85,B 0,C 180,E1 -23643.103,E2 -23643.103} C_VEL
LIN {X 0,Y 163.537,Z 750.418,A -85,B 0,C 180,E1 -23646.575,E2 -23646.575} C_VEL
LIN {X 0,Y 161.08,Z 755.248,A -85,B 0,C 180,E1 -23649.569,E2 -23649.569} C_VEL
LIN {X 0,Y 158.73,Z 759.936,A -85,B 0,C 180,E1 -23653.272,E2 -23653.272} C_VEL
LIN {X 0,Y 156.934,Z 763.518,A -85,B 0,C 180,E1 -23657.059,E2 -23657.059} C_VEL
LIN {X 0,Y 156.087,Z 765.366,A -85,B 0,C 180,E1 -23659.622,E2 -23659.622} C_VEL
LIN {X 0,Y 155.507,Z 766.754,A -85,B 0,C 180,E1 -23662.205,E2 -23662.205} C_VEL
LIN {X 0,Y 154.905,Z 768.348,A -85,B 0,C 180,E1 -23667.397,E2 -23667.397} C_VEL
LIN {X 0,Y 154.861,Z 768.575,A -85,B 0,C 180,E1 -23669.998,E2 -23669.998} C_VEL
LIN {X 0,Y 154.952,Z 768.169,A -85,B 0,C 180,E1 -23673.768,E2 -23673.768} C_VEL
LIN {X 0,Y 155.505,Z 766.831,A -85,B 0,C 180,E1 -23677.79,E2 -23677.79} C_VEL
LIN {X 0,Y 156.085,Z 765.476,A -85,B 0,C 180,E1 -23680.374,E2 -23680.374} C_VEL
LIN {X 0,Y 157.443,Z 762.606,A -85,B 0,C 180,E1 -23684.21,E2 -23684.21} C_VEL
LIN {X 0,Y 159.421,Z 758.71,A -85,B 0,C 180,E1 -23687.972,E2 -23687.972} C_VEL
LIN {X 0,Y 161.951,Z 753.689,A -85,B 0,C 180,E1 -23691.643,E2 -23691.643} C_VEL
LIN {X 0,Y 165.13,Z 747.359,A -85,B 0,C 180,E1 -23695.186,E2 -23695.186} C_VEL
LIN {X 0,Y 168.755,Z 739.637,A -85,B 0,C 180,E1 -23698.521,E2 -23698.521} C_VEL
LIN {X 0,Y 172.095,Z 731.543,A -85,B 0,C 180,E1 -23701.307,E2 -23701.307} C_VEL
LIN {X 0,Y 175.922,Z 721.509,A -85,B 0,C 180,E1 -23704.004,E2 -23704.004} C_VEL
LIN {X 0,Y 179.722,Z 710.404,A -85,B 0,C 180,E1 -23706.258,E2 -23706.258} C_VEL
LIN {X 0,Y 182.78,Z 699.513,A -85,B 0,C 180,E1 -23707.964,E2 -23707.964} C_VEL
LIN {X 0,Y 185.476,Z 687.464,A -85,B 0,C 180,E1 -23709.394,E2 -23709.394} C_VEL
LIN {X 0,Y 187.624,Z 674.861,A -85,B 0,C 180,E1 -23710.443,E2 -23710.443} C_VEL
LIN {X 0,Y 189.024,Z 661.437,A -85,B 0,C 180,E1 -23711.156,E2 -23711.156} C_VEL
LIN {X 0,Y 191.474,Z 620.404,A -85,B 0,C 180,E1 -23712.556,E2 -23712.556} C_VEL
LIN {X 0,Y 186.102,Z 607.603,A -85,B 0,C 180,E1 -23714.784,E2 -23714.784} C_VEL
LIN {X 0,Y 180.158,Z 597.419,A -85,B 0,C 180,E1 -23717.289,E2 -23717.289} C_VEL
LIN {X 0,Y 173.978,Z 587.868,A -85,B 0,C 180,E1 -23720.159,E2 -23720.159} C_VEL
LIN {X 0,Y 170.639,Z 583.177,A -85,B 0,C 180,E1 -23721.844,E2 -23721.844} C_VEL
LIN {X 0,Y 168.182,Z 579.695,A -85,B 0,C 180,E1 -23723.173,E2 -23723.173} C_VEL
LIN {X 0,Y 165.463,Z 575.899,A -85,B 0,C 180,E1 -23724.738,E2 -23724.738} C_VEL
LIN {X 0,Y 162.368,Z 572.443,A -85,B 0,C 180,E1 -23726.597,E2 -23726.597} C_VEL
LIN {X 0,Y 161.266,Z 570.418,A -85,B 0,C 180,E1 -23727.363,E2 -23727.363} C_VEL
LIN {X 0,Y 158.941,Z 568.522,A -85,B 0,C 180,E1 -23728.869,E2 -23728.869} C_VEL
LIN {X 0,Y 157.608,Z 566.244,A -85,B 0,C 180,E1 -23729.89,E2 -23729.89} C_VEL
LIN {X 0,Y 157.283,Z 564.891,A -85,B 0,C 180,E1 -23730.283,E2 -23730.283} C_VEL
LIN {X 0,Y 157.316,Z 564.877,A -85,B 0,C 180,E1 -23733.465,E2 -23733.465} C_VEL
LIN {X 0,Y 157.389,Z 564.87,A -85,B 0,C 180,E1 -23739.665,E2 -23739.665} C_VEL
LIN {X 0,Y 157.463,Z 564.85,A -85,B 0,C 180,E1 -23744.467,E2 -23744.467} C_VEL
LIN {X 0,Y 157.723,Z 564.815,A -85,B 0,C 180,E1 -23749.733,E2 -23749.733} C_VEL
LIN {X 0,Y 157.805,Z 564.818,A -85,B 0,C 180,E1 -23752.322,E2 -23752.322} C_VEL
LIN {X 0,Y 158.253,Z 564.773,A -85,B 0,C 180,E1 -23760,E2 -23760} C_VEL
LIN {X 0,Y 157.818,Z 564.822,A -85,B 0,C 180,E1 -23767.677,E2 -23767.677} C_VEL
LIN {X 0,Y 157.699,Z 564.824,A -85,B 0,C 180,E1 -23771.361,E2 -23771.361} C_VEL
LIN {X 0,Y 157.463,Z 564.852,A -85,B 0,C 180,E1 -23775.533,E2 -23775.533} C_VEL
LIN {X 0,Y 157.365,Z 564.869,A -85,B 0,C 180,E1 -23780.933,E2 -23780.933} C_VEL
LIN {X 0,Y 157.308,Z 564.877,A -85,B 0,C 180,E1 -23786.685,E2 -23786.685} C_VEL
LIN {X 0,Y 157.284,Z 564.891,A -85,B 0,C 180,E1 -23789.348,E2 -23789.348} C_VEL
LIN {X 0,Y 158.226,Z 567.611,A -85,B 0,C 180,E1 -23790.256,E2 -23790.256} C_VEL
LIN {X 0,Y 160.375,Z 569.876,A -85,B 0,C 180,E1 -23791.727,E2 -23791.727} C_VEL
LIN {X 0,Y 161.465,Z 570.664,A -85,B 0,C 180,E1 -23792.406,E2 -23792.406} C_VEL
LIN {X 0,Y 163.42,Z 573.892,A -85,B 0,C 180,E1 -23793.714,E2 -23793.714} C_VEL
LIN {X 0,Y 165.554,Z 576.058,A -85,B 0,C 180,E1 -23794.958,E2 -23794.958} C_VEL
LIN {X 0,Y 169.847,Z 582.806,A -85,B 0,C 180,E1 -23797.427,E2 -23797.427} C_VEL
LIN {X 0,Y 172.979,Z 587.933,A -85,B 0,C 180,E1 -23799.084,E2 -23799.084} C_VEL
LIN {X 0,Y 177.542,Z 595.954,A -85,B 0,C 180,E1 -23801.334,E2 -23801.334} C_VEL
LIN {X 0,Y 183.07,Z 607.056,A -85,B 0,C 180,E1 -23803.87,E2 -23803.87} C_VEL
LIN {X 0,Y 188.701,Z 620.549,A -85,B 0,C 180,E1 -23806.308,E2 -23806.308} C_VEL
LIN {X 0,Y 190.741,Z 626.334,A -85,B 0,C 180,E1 -23807.177,E2 -23807.177} C_VEL
LIN {X 0,Y 190.961,Z 630.403,A -85,B 0,C 180,E1 -23807.441,E2 -23807.441} C_VEL
LIN {X 0,Y 188.189,Z 673.961,A -85,B 0,C 180,E1 -23808.95,E2 -23808.95} C_VEL
LIN {X 0,Y 186.499,Z 687.113,A -85,B 0,C 180,E1 -23809.765,E2 -23809.765} C_VEL
LIN {X 0,Y 183.893,Z 699.915,A -85,B 0,C 180,E1 -23810.909,E2 -23810.909} C_VEL
LIN {X 0,Y 181.049,Z 711.001,A -85,B 0,C 180,E1 -23812.313,E2 -23812.313} C_VEL
LIN {X 0,Y 177.77,Z 721.65,A -85,B 0,C 180,E1 -23814.088,E2 -23814.088} C_VEL
LIN {X 0,Y 175.653,Z 726.519,A -85,B 0,C 180,E1 -23814.963,E2 -23814.963} C_VEL
LIN {X 0,Y 170.378,Z 734.027,A -85,B 0,C 180,E1 -23816.211,E2 -23816.211} C_VEL
LIN {X 0,Y 164.874,Z 741.025,A -85,B 0,C 180,E1 -23817.699,E2 -23817.699} C_VEL
LIN {X 0,Y 162.454,Z 745.045,A -85,B 0,C 180,E1 -23818.946,E2 -23818.946} C_VEL
LIN {X 0,Y 158.856,Z 752.858,A -85,B 0,C 180,E1 -23822.14,E2 -23822.14} C_VEL
LIN {X 0,Y 155.218,Z 760.062,A -85,B 0,C 180,E1 -23825.955,E2 -23825.955} C_VEL
LIN {X 0,Y 152.368,Z 765.58,A -85,B 0,C 180,E1 -23829.764,E2 -23829.764} C_VEL
LIN {X 0,Y 150.14,Z 769.913,A -85,B 0,C 180,E1 -23833.691,E2 -23833.691} C_VEL
LIN {X 0,Y 149.14,Z 772.215,A -85,B 0,C 180,E1 -23836.375,E2 -23836.375} C_VEL
LIN {X 0,Y 148.391,Z 774.078,A -85,B 0,C 180,E1 -23839.082,E2 -23839.082} C_VEL
LIN {X 0,Y 147.898,Z 775.476,A -85,B 0,C 180,E1 -23841.807,E2 -23841.807} C_VEL
LIN {X 0,Y 147.634,Z 776.475,A -85,B 0,C 180,E1 -23844.539,E2 -23844.539} C_VEL
LIN {X 0,Y 147.622,Z 777.234,A -85,B 0,C 180,E1 -23848.775,E2 -23848.775} C_VEL
LIN {X 0,Y 147.839,Z 776.966,A -85,B 0,C 180,E1 -23853.34,E2 -23853.34} C_VEL
LIN {X 0,Y 148.702,Z 775.459,A -85,B 0,C 180,E1 -23858.154,E2 -23858.154} C_VEL
LIN {X 0,Y 150.668,Z 772.662,A -85,B 0,C 180,E1 -23863.146,E2 -23863.146} C_VEL
LIN {X 0,Y 152.454,Z 776.815,A -85,B 0,C 180,E1 -23867.439,E2 -23867.439} C_VEL
LIN {X 0,Y 155.027,Z 779.584,A -85,B 0,C 180,E1 -23871.267,E2 -23871.267} C_VEL
LIN {X 0,Y 157.183,Z 780.947,A -85,B 0,C 180,E1 -23873.731,E2 -23873.731} C_VEL
LIN {X 0,Y 159.856,Z 781.808,A -85,B 0,C 180,E1 -23876.084,E2 -23876.084} C_VEL
LIN {X 0,Y 166.486,Z 782.438,A -85,B 0,C 180,E1 -23880.438,E2 -23880.438} C_VEL
LIN {X 0,Y 170.291,Z 782.097,A -85,B 0,C 180,E1 -23882.449,E2 -23882.449} C_VEL
LIN {X 0,Y 174.399,Z 781.263,A -85,B 0,C 180,E1 -23884.347,E2 -23884.347} C_VEL
LIN {X 0,Y 183.42,Z 778.374,A -85,B 0,C 180,E1 -23887.813,E2 -23887.813} C_VEL
LIN {X 0,Y 190.756,Z 774.878,A -85,B 0,C 180,E1 -23890.149,E2 -23890.149} C_VEL
LIN {X 0,Y 198.678,Z 770.2,A -85,B 0,C 180,E1 -23892.232,E2 -23892.232} C_VEL
LIN {X 0,Y 207.234,Z 763.941,A -85,B 0,C 180,E1 -23894.15,E2 -23894.15} C_VEL
LIN {X 0,Y 214.279,Z 757.717,A -85,B 0,C 180,E1 -23895.511,E2 -23895.511} C_VEL
LIN {X 0,Y 215.781,Z 756.232,A -85,B 0,C 180,E1 -23895.772,E2 -23895.772} C_VEL
LIN {X 0,Y 213.972,Z 758.06,A -85,B 0,C 180,E1 -23896.389,E2 -23896.389} C_VEL
LIN {X 0,Y 205.272,Z 765.631,A -85,B 0,C 180,E1 -23898.115,E2 -23898.115} C_VEL
LIN {X 0,Y 196.98,Z 771.417,A -85,B 0,C 180,E1 -23900.043,E2 -23900.043} C_VEL
LIN {X 0,Y 189.151,Z 775.784,A -85,B 0,C 180,E1 -23902.188,E2 -23902.188} C_VEL
LIN {X 0,Y 181.879,Z 778.742,A -85,B 0,C 180,E1 -23904.576,E2 -23904.576} C_VEL
LIN {X 0,Y 177.345,Z 780.158,A -85,B 0,C 180,E1 -23906.303,E2 -23906.303} C_VEL
LIN {X 0,Y 173.01,Z 781.041,A -85,B 0,C 180,E1 -23908.124,E2 -23908.124} C_VEL
LIN {X 0,Y 168.947,Z 781.413,A -85,B 0,C 180,E1 -23910.054,E2 -23910.054} C_VEL
LIN {X 0,Y 165.256,Z 781.363,A -85,B 0,C 180,E1 -23912.108,E2 -23912.108} C_VEL
LIN {X 0,Y 161.872,Z 780.893,A -85,B 0,C 180,E1 -23914.267,E2 -23914.267} C_VEL
LIN {X 0,Y 158.91,Z 779.957,A -85,B 0,C 180,E1 -23916.544,E2 -23916.544} C_VEL
LIN {X 0,Y 156.407,Z 778.522,A -85,B 0,C 180,E1 -23918.932,E2 -23918.932} C_VEL
LIN {X 0,Y 153.458,Z 775.62,A -85,B 0,C 180,E1 -23922.681,E2 -23922.681} C_VEL
LIN {X 0,Y 151.419,Z 771.635,A -85,B 0,C 180,E1 -23926.581,E2 -23926.581} C_VEL
LIN {X 0,Y 150.33,Z 765.84,A -85,B 0,C 180,E1 -23930.922,E2 -23930.922} C_VEL
LIN {X 0,Y 150.295,Z 759.773,A -85,B 0,C 180,E1 -23934.634,E2 -23934.634} C_VEL
LIN {X 0,Y 150.599,Z 752.756,A -85,B 0,C 180,E1 -23937.994,E2 -23937.994} C_VEL
LIN {X 0,Y 150.935,Z 745.724,A -85,B 0,C 180,E1 -23940.667,E2 -23940.667} C_VEL
LIN {X 0,Y 151.259,Z 736.996,A -85,B 0,C 180,E1 -23943.33,E2 -23943.33} C_VEL
LIN {X 0,Y 151.495,Z 727.172,A -85,B 0,C 180,E1 -23945.658,E2 -23945.658} C_VEL
LIN {X 0,Y 151.897,Z 715.987,A -85,B 0,C 180,E1 -23947.644,E2 -23947.644} C_VEL
LIN {X 0,Y 152.174,Z 703.636,A -85,B 0,C 180,E1 -23949.219,E2 -23949.219} C_VEL
LIN {X 0,Y 152.415,Z 657.498,A -85,B 0,C 180,E1 -23953.59,E2 -23953.59} C_VEL
LIN {X 0,Y 150.925,Z 634.456,A -85,B 0,C 180,E1 -23955.559,E2 -23955.559} C_VEL
LIN {X 0,Y 150.79,Z 632.067,A -85,B 0,C 180,E1 -23955.906,E2 -23955.906} C_VEL
LIN {X 0,Y 152.952,Z 604.891,A -85,B 0,C 180,E1 -23965.153,E2 -23965.153} C_VEL
LIN {X 0,Y 154.642,Z 591.929,A -85,B 0,C 180,E1 -23969.62,E2 -23969.62} C_VEL
LIN {X 0,Y 155.116,Z 590.264,A -85,B 0,C 180,E1 -23970.672,E2 -23970.672} C_VEL
LIN {X 0,Y 155.546,Z 590.294,A -85,B 0,C 180,E1 -23971.185,E2 -23971.185} C_VEL
LIN {X 0,Y 157.427,Z 590.632,A -85,B 0,C 180,E1 -23972.393,E2 -23972.393} C_VEL
LIN {X 0,Y 159.594,Z 589.314,A -85,B 0,C 180,E1 -23973.503,E2 -23973.503} C_VEL
LIN {X 0,Y 163.432,Z 589.241,A -85,B 0,C 180,E1 -23975.495,E2 -23975.495} C_VEL
LIN {X 0,Y 165.554,Z 588.451,A -85,B 0,C 180,E1 -23976.464,E2 -23976.464} C_VEL
LIN {X 0,Y 167.366,Z 588.697,A -85,B 0,C 180,E1 -23977.32,E2 -23977.32} C_VEL
LIN {X 0,Y 171.54,Z 594.727,A -85,B 0,C 180,E1 -23979.518,E2 -23979.518} C_VEL
LIN {X 0,Y 177.65,Z 604.584,A -85,B 0,C 180,E1 -23982.452,E2 -23982.452} C_VEL
LIN {X 0,Y 182.174,Z 612.96,A -85,B 0,C 180,E1 -23984.463,E2 -23984.463} C_VEL
LIN {X 0,Y 186.035,Z 622.346,A -85,B 0,C 180,E1 -23986.167,E2 -23986.167} C_VEL
LIN {X 0,Y 183.242,Z 665.732,A -85,B 0,C 180,E1 -23987.71,E2 -23987.71} C_VEL
LIN {X 0,Y 181.476,Z 678.872,A -85,B 0,C 180,E1 -23988.522,E2 -23988.522} C_VEL
LIN {X 0,Y 179.221,Z 691.012,A -85,B 0,C 180,E1 -23989.679,E2 -23989.679} C_VEL
LIN {X 0,Y 176.458,Z 702.285,A -85,B 0,C 180,E1 -23991.147,E2 -23991.147} C_VEL
LIN {X 0,Y 172.803,Z 713.91,A -85,B 0,C 180,E1 -23993.136,E2 -23993.136} C_VEL
LIN {X 0,Y 168.965,Z 724.352,A -85,B 0,C 180,E1 -23995.476,E2 -23995.476} C_VEL
LIN {X 0,Y 164.949,Z 734.119,A -85,B 0,C 180,E1 -23998.339,E2 -23998.339} C_VEL
LIN {X 0,Y 161.36,Z 742.114,A -85,B 0,C 180,E1 -24001.371,E2 -24001.371} C_VEL
LIN {X 0,Y 157.657,Z 749.513,A -85,B 0,C 180,E1 -24004.943,E2 -24004.943} C_VEL
LIN {X 0,Y 154.432,Z 755.455,A -85,B 0,C 180,E1 -24008.647,E2 -24008.647} C_VEL
LIN {X 0,Y 151.953,Z 760.142,A -85,B 0,C 180,E1 -24012.502,E2 -24012.502} C_VEL
LIN {X 0,Y 150.019,Z 763.724,A -85,B 0,C 180,E1 -24016.451,E2 -24016.451} C_VEL
LIN {X 0,Y 149.113,Z 765.572,A -85,B 0,C 180,E1 -24019.131,E2 -24019.131} C_VEL
LIN {X 0,Y 148.47,Z 766.959,A -85,B 0,C 180,E1 -24021.833,E2 -24021.833} C_VEL
LIN {X 0,Y 147.855,Z 768.43,A -85,B 0,C 180,E1 -24026.564,E2 -24026.564} C_VEL
LIN {X 0,Y 147.766,Z 768.78,A -85,B 0,C 180,E1 -24029.998,E2 -24029.998} C_VEL
LIN {X 0,Y 147.839,Z 768.479,A -85,B 0,C 180,E1 -24033.335,E2 -24033.335} C_VEL
LIN {X 0,Y 148.468,Z 767.036,A -85,B 0,C 180,E1 -24038.162,E2 -24038.162} C_VEL
LIN {X 0,Y 149.11,Z 765.68,A -85,B 0,C 180,E1 -24040.865,E2 -24040.865} C_VEL
LIN {X 0,Y 150.572,Z 762.809,A -85,B 0,C 180,E1 -24044.873,E2 -24044.873} C_VEL
LIN {X 0,Y 152.693,Z 758.913,A -85,B 0,C 180,E1 -24048.793,E2 -24048.793} C_VEL
LIN {X 0,Y 155.379,Z 753.892,A -85,B 0,C 180,E1 -24052.608,E2 -24052.608} C_VEL
LIN {X 0,Y 158.746,Z 747.561,A -85,B 0,C 180,E1 -24056.275,E2 -24056.275} C_VEL
LIN {X 0,Y 162.414,Z 740.116,A -85,B 0,C 180,E1 -24059.611,E2 -24059.611} C_VEL
LIN {X 0,Y 166.151,Z 731.569,A -85,B 0,C 180,E1 -24062.633,E2 -24062.633} C_VEL
LIN {X 0,Y 170.081,Z 721.71,A -85,B 0,C 180,E1 -24065.342,E2 -24065.342} C_VEL
LIN {X 0,Y 174.06,Z 710.604,A -85,B 0,C 180,E1 -24067.637,E2 -24067.637} C_VEL
LIN {X 0,Y 177.241,Z 699.712,A -85,B 0,C 180,E1 -24069.375,E2 -24069.375} C_VEL
LIN {X 0,Y 180.063,Z 687.661,A -85,B 0,C 180,E1 -24070.823,E2 -24070.823} C_VEL
LIN {X 0,Y 182.284,Z 675.059,A -85,B 0,C 180,E1 -24071.889,E2 -24071.889} C_VEL
LIN {X 0,Y 183.77,Z 661.261,A -85,B 0,C 180,E1 -24072.626,E2 -24072.626} C_VEL
LIN {X 0,Y 186.188,Z 622.57,A -85,B 0,C 180,E1 -24073.964,E2 -24073.964} C_VEL
LIN {X 0,Y 181.675,Z 611.757,A -85,B 0,C 180,E1 -24075.963,E2 -24075.963} C_VEL
LIN {X 0,Y 175.404,Z 600.761,A -85,B 0,C 180,E1 -24078.806,E2 -24078.806} C_VEL
LIN {X 0,Y 170.038,Z 592.506,A -85,B 0,C 180,E1 -24081.478,E2 -24081.478} C_VEL
LIN {X 0,Y 165.142,Z 585.432,A -85,B 0,C 180,E1 -24084.194,E2 -24084.194} C_VEL
LIN {X 0,Y 162.073,Z 581.254,A -85,B 0,C 180,E1 -24086.061,E2 -24086.061} C_VEL
LIN {X 0,Y 159.438,Z 577.999,A -85,B 0,C 180,E1 -24087.775,E2 -24087.775} C_VEL
LIN {X 0,Y 158.547,Z 576.618,A -85,B 0,C 180,E1 -24088.411,E2 -24088.411} C_VEL
LIN {X 0,Y 155.998,Z 573.953,A -85,B 0,C 180,E1 -24090.222,E2 -24090.222} C_VEL
LIN {X 0,Y 154.688,Z 571.496,A -85,B 0,C 180,E1 -24091.321,E2 -24091.321} C_VEL
LIN {X 0,Y 152.117,Z 569.719,A -85,B 0,C 180,E1 -24093.343,E2 -24093.343} C_VEL
LIN {X 0,Y 150.618,Z 567.324,A -85,B 0,C 180,E1 -24094.775,E2 -24094.775} C_VEL
LIN {X 0,Y 150.247,Z 565.769,A -85,B 0,C 180,E1 -24095.287,E2 -24095.287} C_VEL
LIN {X 0,Y 150.36,Z 565.755,A -85,B 0,C 180,E1 -24100.902,E2 -24100.902} C_VEL
LIN {X 0,Y 150.448,Z 565.742,A -85,B 0,C 180,E1 -24106.493,E2 -24106.493} C_VEL
LIN {X 0,Y 150.645,Z 565.698,A -85,B 0,C 180,E1 -24109.245,E2 -24109.245} C_VEL
LIN {X 0,Y 150.739,Z 565.693,A -85,B 0,C 180,E1 -24111.959,E2 -24111.959} C_VEL
LIN {X 0,Y 151.213,Z 565.649,A -85,B 0,C 180,E1 -24120,E2 -24120} C_VEL
LIN {X 0,Y 150.757,Z 565.696,A -85,B 0,C 180,E1 -24128.039,E2 -24128.039} C_VEL
LIN {X 0,Y 150.628,Z 565.705,A -85,B 0,C 180,E1 -24131.545,E2 -24131.545} C_VEL
LIN {X 0,Y 150.368,Z 565.735,A -85,B 0,C 180,E1 -24136.286,E2 -24136.286} C_VEL
LIN {X 0,Y 150.346,Z 565.743,A -85,B 0,C 180,E1 -24140.794,E2 -24140.794} C_VEL
LIN {X 0,Y 150.251,Z 565.771,A -85,B 0,C 180,E1 -24144.343,E2 -24144.343} C_VEL
LIN {X 0,Y 150.963,Z 568.145,A -85,B 0,C 180,E1 -24145.232,E2 -24145.232} C_VEL
LIN {X 0,Y 152.896,Z 570.412,A -85,B 0,C 180,E1 -24146.946,E2 -24146.946} C_VEL
LIN {X 0,Y 154.763,Z 571.669,A -85,B 0,C 180,E1 -24148.385,E2 -24148.385} C_VEL
LIN {X 0,Y 156.509,Z 574.692,A -85,B 0,C 180,E1 -24149.812,E2 -24149.812} C_VEL
LIN {X 0,Y 158.954,Z 577.11,A -85,B 0,C 180,E1 -24151.509,E2 -24151.509} C_VEL
LIN {X 0,Y 161.394,Z 580.608,A -85,B 0,C 180,E1 -24153.164,E2 -24153.164} C_VEL
LIN {X 0,Y 162.927,Z 582.358,A -85,B 0,C 180,E1 -24154.109,E2 -24154.109} C_VEL
LIN {X 0,Y 166.852,Z 588.671,A -85,B 0,C 180,E1 -24156.486,E2 -24156.486} C_VEL
LIN {X 0,Y 171.466,Z 596.574,A -85,B 0,C 180,E1 -24159.026,E2 -24159.026} C_VEL
LIN {X 0,Y 177.334,Z 608.089,A -85,B 0,C 180,E1 -24161.981,E2 -24161.981} C_VEL
LIN {X 0,Y 182.456,Z 620.208,A -85,B 0,C 180,E1 -24164.397,E2 -24164.397} C_VEL
LIN {X 0,Y 185.647,Z 628.74,A -85,B 0,C 180,E1 -24165.839,E2 -24165.839} C_VEL
LIN {X 0,Y 185.6,Z 633.596,A -85,B 0,C 180,E1 -24166.08,E2 -24166.08} C_VEL
LIN {X 0,Y 182.905,Z 673.812,A -85,B 0,C 180,E1 -24167.495,E2 -24167.495} C_VEL
LIN {X 0,Y 181.03,Z 687.598,A -85,B 0,C 180,E1 -24168.367,E2 -24168.367} C_VEL
LIN {X 0,Y 178.447,Z 699.717,A -85,B 0,C 180,E1 -24169.473,E2 -24169.473} C_VEL
LIN {X 0,Y 175.488,Z 710.801,A -85,B 0,C 180,E1 -24170.897,E2 -24170.897} C_VEL
LIN {X 0,Y 171.762,Z 722.354,A -85,B 0,C 180,E1 -24172.88,E2 -24172.88} C_VEL
LIN {X 0,Y 167.816,Z 732.759,A -85,B 0,C 180,E1 -24175.211,E2 -24175.211} C_VEL
LIN {X 0,Y 164.168,Z 741.271,A -85,B 0,C 180,E1 -24177.651,E2 -24177.651} C_VEL
LIN {X 0,Y 162.454,Z 745.045,A -85,B 0,C 180,E1 -24178.946,E2 -24178.946} C_VEL
LIN {X 0,Y 160.069,Z 748.912,A -85,B 0,C 180,E1 -24180.306,E2 -24180.306} C_VEL
LIN {X 0,Y 154.611,Z 754.713,A -85,B 0,C 180,E1 -24182.467,E2 -24182.467} C_VEL
LIN {X 0,Y 149.271,Z 759.915,A -85,B 0,C 180,E1 -24184.944,E2 -24184.944} C_VEL
LIN {X 0,Y 147.137,Z 762.745,A -85,B 0,C 180,E1 -24186.772,E2 -24186.772} C_VEL
